// TIA Portal project "Arenas_Pantoja_Ospina_PF" (V15)
// Vorlageprojekt für das Buch mit Zielsystem S7-1200

(* hardware
DEVICE "S7-1200-Station_1"  S7-1200 Station
   slot 0: "Baugruppenträger_0"  Rack  V1.0
   slot 1: "PLC_1"  CPU 1214C AC/DC/Rly  6ES7 214-1BG40-0XB0  V4.1
*)

// ===== PLC "PLC_1"  CPU 1214C AC/DC/Rly =====

VAR_GLOBAL   // PLC tag table "Standard-Variablentabelle"
   "START" AT %E0.0 : Bool;
   "M200" AT %M200.0 : Bool;
   "P0" AT %M0.0 : Bool;
   "AUTOMATICO" AT %I6.0 : Bool;
   "MANUAL" AT %I6.1 : Bool;
   "P1" AT %M0.1 : Bool;
   "AAAAAAAAAAAAAAAAAAAAAAAAAAAAAAAAAAA" AT %M40.0 : Bool;
   "P2" AT %M0.2 : Bool;
   "I1_EntradaObjetos" AT %I0.1 : Bool;
   "P3" AT %M0.3 : Bool;
   "I2_SensorPasoInicial" AT %I0.2 : Bool;
   "FP_I2_SensorPasoInicial" AT %M50.0 : Bool;
   "P4" AT %M0.4 : Bool;
   "FN_I2_SensorPasoInicial" AT %M50.1 : Bool;
   "P5" AT %M0.5 : Bool;
   "I3_SensorVisionBR" AT %I0.3 : Bool;
   "I4_SensorVisionGR" AT %I0.4 : Bool;
   "I5_SensorVisionBG" AT %I0.5 : Bool;
   "P6" AT %M0.6 : Bool;
   "I6_BandaBascula" AT %I0.6 : Bool;
   "FP_I6_BandaBascula(1)" AT %M50.2 : Bool;
   "P7" AT %M0.7 : Bool;
   "P8" AT %M1.0 : Bool;
   "FP_I8_SensorLeft" AT %M50.3 : Bool;
   "I8_SensorLeft" AT %I1.0 : Bool;
   "FN_I8_SensorLeft" AT %M50.4 : Bool;
   "P9" AT %M1.1 : Bool;
   "P10" AT %M1.2 : Bool;
   "FP_I6_BandaBascula_2" AT %M50.5 : Bool;
   "P11" AT %M1.3 : Bool;
   "I7_SensorForward" AT %I0.7 : Bool;
   "FP_I7_SensorForward" AT %M50.6 : Bool;
   "P12" AT %M1.4 : Bool;
   "FN_I7_SensorForward_3" AT %M50.7 : Bool;
   "P13" AT %M1.5 : Bool;
   "P14" AT %M1.6 : Bool;
   "FP_I6_BandaBascula_3" AT %M51.0 : Bool;
   "P15" AT %M1.7 : Bool;
   "I9_SensorRigth" AT %I1.1 : Bool;
   "P16" AT %M2.0 : Bool;
   "FP_I9_SensorRigth" AT %M51.1 : Bool;
   "FN_I9_SensorRigth_2" AT %M51.2 : Bool;
   "P17" AT %M2.1 : Bool;
   "Q0_EntradaObjetos" AT %Q0.0 : Bool;
   "Q1_BandaInicial" AT %Q0.1 : Bool;
   "Q2_BandaInicial2" AT %Q0.2 : Bool;
   "Q3_Forward" AT %Q0.3 : Bool;
   "Q4_Left" AT %Q0.4 : Bool;
   "Q5_Right" AT %Q0.5 : Bool;
   "Q6_BandaLeft1" AT %Q0.6 : Bool;
   "Q7_BandaForward1" AT %Q0.7 : Bool;
   "Q8_BandaRigth1" AT %Q1.0 : Bool;
   "Tag_2" AT %MD0 : DWord;
   "I10_SensorLeft2" AT %I1.2 : Bool;
   "FP_I10_SensorLeft2" AT %M51.3 : Bool;
   "P18" AT %M2.2 : Bool;
   "P19" AT %M2.3 : Bool;
   "FN_I10_SensorLeft2" AT %M51.4 : Bool;
   "P20" AT %M2.4 : Bool;
   "I13_SensorLeft3" AT %I1.5 : Bool;
   "FP_I13_SensorLeft3" AT %M51.5 : Bool;
   "FN_I13_SensorLeft3" AT %M51.6 : Bool;
   "P21" AT %M2.5 : Bool;
   "P22" AT %M2.6 : Bool;
   "I11_SensorForward2" AT %I1.3 : Bool;
   "FP_I11_SensorForward2" AT %M51.7 : Bool;
   "P23" AT %M2.7 : Bool;
   "FN_I11_SensorForward2" AT %M52.0 : Bool;
   "P24" AT %M3.0 : Bool;
   "I14_SensorForward3" AT %I1.6 : Bool;
   "FP_I14_SensorForward3" AT %M52.1 : Bool;
   "P25" AT %M3.1 : Bool;
   "I12_SensorRigth2" AT %I1.4 : Bool;
   "FP_I12_SensorRigth2" AT %M52.2 : Bool;
   "P26" AT %M3.2 : Bool;
   "FN_I12_SensorRigth2" AT %M52.3 : Bool;
   "P27" AT %M3.3 : Bool;
   "P28" AT %M3.4 : Bool;
   "I15_SensorRigth3" AT %I1.7 : Bool;
   "FP_I15_SensorRigth3" AT %M52.4 : Bool;
   "P29" AT %M3.5 : Bool;
   "FN_I15_SensorRigth3" AT %M52.5 : Bool;
   "Q9_BandaLeft2" AT %Q1.1 : Bool;
   "Q10_BandaForward2" AT %Q1.2 : Bool;
   "Q11_BandaRigtht2" AT %Q1.3 : Bool;
   "Q12_BandaLeft3" AT %Q1.4 : Bool;
   "Q13_BandaForward3" AT %Q1.5 : Bool;
   "Q14_BandaRigth3" AT %Q1.6 : Bool;
   "Q17_PickZ1" AT %Q2.1 : Bool;
   "Q20_PickZ2" AT %Q2.4 : Bool;
   "Q23_PickZ3" AT %Q2.7 : Bool;
   "FN_I14_SensorForward3" AT %M52.6 : Bool;
   "P30" AT %M3.6 : Bool;
   "I16_SensorGrab1" AT %I2.0 : Bool;
   "FP_I16_SensorGrab1" AT %M52.7 : Bool;
   "P31" AT %M3.7 : Bool;
   "P32" AT %M4.0 : Bool;
   "P33" AT %M4.1 : Bool;
   "P34" AT %M4.2 : Bool;
   "P35" AT %M4.3 : Bool;
   "Q15_PickX1" AT %Q1.7 : Bool;
   "Q16_PickGrab1" AT %Q2.0 : Bool;
   "I17_SensorGrab2" AT %I2.1 : Bool;
   "FP_I17_SensorGrab1" AT %M53.0 : Bool;
   "P36" AT %M4.4 : Bool;
   "P37" AT %M4.5 : Bool;
   "P38" AT %M4.6 : Bool;
   "P39" AT %M4.7 : Bool;
   "P40" AT %M5.0 : Bool;
   "P41" AT %M5.1 : Bool;
   "Q18_PickX2" AT %Q2.2 : Bool;
   "Q19_PickGrab2" AT %Q2.3 : Bool;
   "I18_SensorGrab3" AT %I2.2 : Bool;
   "FP_I18_SensorGrab3" AT %M53.1 : Bool;
   "P42" AT %M5.2 : Bool;
   "P43" AT %M5.3 : Bool;
   "P44" AT %M5.4 : Bool;
   "P45" AT %M5.5 : Bool;
   "P46" AT %M5.6 : Bool;
   "P47" AT %M5.7 : Bool;
   "Q21_PickX3" AT %Q2.5 : Bool;
   "Q22_PickGrab3" AT %Q2.6 : Bool;
   "I19_SensorBandaA1" AT %I2.3 : Bool;
   "FP_I19_SensorBandaA1" AT %M53.2 : Bool;
   "P48" AT %M6.0 : Bool;
   "I20_SensorBandaA2" AT %I2.4 : Bool;
   "FP_I20_SensorBandaA2" AT %M53.3 : Bool;
   "P49" AT %M6.1 : Bool;
   "I21_SensorBandaA3" AT %I2.5 : Bool;
   "FP_21_SensorBandaA3" AT %M53.4 : Bool;
   "P50" AT %M6.2 : Bool;
   "Q24_BandaLeftA1" AT %Q3.0 : Bool;
   "Q25_BandaLeftA2" AT %Q3.1 : Bool;
   "Q26_BandaForwardA1" AT %Q3.2 : Bool;
   "Q27_BandaForwardA2" AT %Q3.3 : Bool;
   "Q28_BandaRightA1" AT %Q3.4 : Bool;
   "Q29_BandaRightA2" AT %Q3.5 : Bool;
   "Q30_EmisorA1" AT %Q3.6 : Bool;
   "Q31_EmisorA2" AT %Q3.7 : Bool;
   "Q32_EmisorA3" AT %Q4.0 : Bool;
   "P51" AT %M6.3 : Bool;
   "I22_LimAdelaA1" AT %I2.6 : Bool;
   "FP_I22_LimAdelaA1" AT %M53.5 : Bool;
   "P52" AT %M6.4 : Bool;
   "I23_LimSubA1" AT %I2.7 : Bool;
   "FP_I23_LimSubA1" AT %M53.6 : Bool;
   "Q33_AdelanteA1" AT %Q4.1 : Bool;
   "Q34_SubirA1" AT %Q4.2 : Bool;
   "P53" AT %M6.5 : Bool;
   "I24_LimAdelaA2" AT %I3.0 : Bool;
   "FP_I24_LimAdelaA2" AT %M53.7 : Bool;
   "P54" AT %M6.6 : Bool;
   "I25_LimSubA2" AT %I3.1 : Bool;
   "FN_I25_LimSubA2" AT %M54.0 : Bool;
   "Q36_AdelanteA2" AT %Q4.4 : Bool;
   "Q37_SubirA2" AT %Q4.5 : Bool;
   "P55" AT %M6.7 : Bool;
   "P56" AT %M7.0 : Bool;
   "Q39_AdelanteA3" AT %Q4.7 : Bool;
   "Q40_SubirA3" AT %Q5.0 : Bool;
   "P57" AT %M7.1 : Bool;
   "P58" AT %M7.2 : Bool;
   "P59" AT %M7.3 : Bool;
   "Right count" AT %QW40 : Int;
   "Tag_4" AT %QW50 : Int;
   "Q41_PosicionA1" AT %QW30 : Int;
   "Tag_6" AT %QW60 : Int;
   "Tag_7" AT %QW90 : Int;
   "Q42_PosicionA2" AT %QW32 : Int;
   "Tag_9" AT %QW33 : Int;
   "Q43_PosicionA3" AT %QW34 : Int;
   "P60" AT %M7.4 : Bool;
   "P61" AT %M7.5 : Bool;
   "P62" AT %M7.6 : Bool;
   "Q35_AtrasA1" AT %Q4.3 : Bool;
   "P63" AT %M7.7 : Bool;
   "P64" AT %M8.0 : Bool;
   "P65" AT %M8.1 : Bool;
   "P66" AT %M8.2 : Bool;
   "P67" AT %M8.3 : Bool;
   "Q38_AtrasA2" AT %Q4.6 : Bool;
   "P68" AT %M8.4 : Bool;
   "P69" AT %M8.5 : Bool;
   "P70" AT %M8.6 : Bool;
   "P71" AT %M8.7 : Bool;
   "Q41_AtrasA3" AT %Q5.1 : Bool;
   "I_4.0_PosicionA1" AT %I4.0 : Bool;
   "FN_I_4.0_PosicionA1" AT %M540.1 : Bool;
   "I_4.1_PosicionA2" AT %I4.1 : Bool;
   "FN_I_4.0_PosicionA1(1)" AT %M54.1 : Bool;
   "FN_I_4.1_PosicionA2" AT %M54.2 : Bool;
   "I_4.2_PosicionA3" AT %I4.2 : Bool;
   "FN_I_4.2_PosicionA3" AT %M54.3 : Bool;
   "P80" AT %M9.0 : Bool;
   "Left count" AT %QW36 : Word;
   "Forward count" AT %QW38 : Int;
   "M.Emitter" AT %I3.2 : Bool;
   "M.BI_B2" AT %I3.3 : Bool;
   "M.Q3_ON" AT %I3.4 : Bool;
   "M.Q3_OFF" AT %I3.5 : Bool;
   "M.LEFT_DECISION" AT %I3.6 : Bool;
   "M.RIGHT_DECISION" AT %I3.7 : Bool;
   "M.Left bands" AT %I4.3 : Bool;
   "M.Forward bands" AT %I4.4 : Bool;
   "M.Right bands" AT %I4.5 : Bool;
   "STOP" AT %I5.7 : Bool;
   "I4.6_M.GrabOn" AT %I4.6 : Bool;
   "I4.7_M.GrabOff" AT %I4.7 : Bool;
   "I5.0_M.EjeXOn" AT %I5.0 : Bool;
   "I5.2_M.EjezOn" AT %I5.2 : Bool;
   "I5.4_M.EmitterM" AT %I5.4 : Bool;
   "I5.1_M.EjeXOff" AT %I5.1 : Bool;
   "I5.3_M.EjezOff" AT %I5.3 : Bool;
   "Q44_LightAutomatico" AT %Q5.2 : Bool;
   "Q45_LightManual" AT %Q5.3 : Bool;
   "I5.5_M.BandasA" AT %I5.5 : Bool;
   "Q46.RemoverM" AT %Q5.4 : Bool;
   "Pin_BL" AT %M10.0 : Bool;
   "ENABLE_BL" AT %M15.0 : Bool;
   "M_Q2_B_LEFT" AT %M20.1 : Bool;
   "M_Q3_B_LEFT" AT %M20.2 : Bool;
   "M_Q4_B_LEFT" AT %M20.3 : Bool;
   "M_Q6_B_LEFT" AT %M20.5 : Bool;
   "M_Q9_B_LEFT" AT %M21.0 : Bool;
   "M_Q12_B_LEFT" AT %M21.3 : Bool;
   "Pout_BL" AT %M10.1 : Bool;
   "Pin_PL" AT %M10.2 : Bool;
   "ENABLE_PL" AT %M15.1 : Bool;
   "M_Q5_B_RIGHT" AT %M20.4 : Bool;
   "M_Q7" AT %M20.6 : Bool;
   "M_Q8_B_RIGHT" AT %M20.7 : Bool;
   "M_Q10" AT %M21.1 : Bool;
   "M_Q11_B_RIGHT" AT %M21.2 : Bool;
   "M_Q13" AT %M21.4 : Bool;
   "M_Q14_B_RIGHT" AT %M21.5 : Bool;
   "M_Q15_P_LEFT" AT %M21.6 : Bool;
   "M_Q16_P_LEFT" AT %M21.7 : Bool;
   "M_Q17_P_LEFT" AT %M22.0 : Bool;
   "M_Q18_B_PF" AT %M22.1 : Bool;
   "M_Q19_B_PF" AT %M22.2 : Bool;
   "M_Q20_B_PF" AT %M22.3 : Bool;
   "M_Q21_P_RIGHT" AT %M22.4 : Bool;
   "M_Q22_P_RIGHT" AT %M22.5 : Bool;
   "M_Q23_P_RIGHT" AT %M22.6 : Bool;
   "M_Q24_G_LEFT" AT %M22.7 : Bool;
   "M_Q25_G_LEFT" AT %M23.0 : Bool;
   "M_Q26_GF" AT %M23.1 : Bool;
   "M_Q27_GF" AT %M23.2 : Bool;
   "M_Q28" AT %M23.3 : Bool;
   "M_Q29" AT %M23.4 : Bool;
   "M_Q30_P_LEFT" AT %M23.5 : Bool;
   "Pout_PL" AT %M10.3 : Bool;
   "P52_Out" AT %M25.0 : Bool;
   "Pin_GL" AT %M10.4 : Bool;
   "ENABLE_GL" AT %M15.2 : Bool;
   "Pout_GL" AT %M10.5 : Bool;
   "M_Q31_B_PF" AT %M23.6 : Bool;
   "M_Q32_P_RIGHT" AT %M23.7 : Bool;
   "M_Q33_G_LEFT" AT %M24.0 : Bool;
   "M_Q34_G_LEFT" AT %M24.1 : Bool;
   "M_Q35_G_LEFT" AT %M24.2 : Bool;
   "M_Q36_GF" AT %M24.3 : Bool;
   "M_Q37_GF" AT %M24.4 : Bool;
   "M_Q38_GF" AT %M24.5 : Bool;
   "M_Q39" AT %M24.6 : Bool;
   "M_Q40" AT %M24.7 : Bool;
   "M_Q41_G_LEFT" AT %M26.0 : Bool;
   "M_Q42_G_FRONT" AT %M26.1 : Bool;
   "P57_Out" AT %M25.1 : Bool;
   "Pin_BF" AT %M10.6 : Bool;
   "ENABLE_BF" AT %M15.3 : Bool;
   "Pout_BF" AT %M10.7 : Bool;
   "M_Q2_B_FRONT" AT %M27.0 : Bool;
   "M_Q3_B_FRONT" AT %M27.1 : Bool;
   "NOHACENADA:D" AT %M27.2 : Bool;
   "M_Q7_B_FRONT" AT %M27.3 : Bool;
   "M_Q10_B_FRONT" AT %M27.4 : Bool;
   "M_Q13_B_FRONT" AT %M27.5 : Bool;
   "Pin_PF" AT %M11.0 : Bool;
   "ENABLE_PF" AT %M15.4 : Bool;
   "Pout_PF" AT %M11.1 : Bool;
   "Pin_GF" AT %M11.2 : Bool;
   "ENABLE_GF" AT %M15.5 : Bool;
   "Pout_GF" AT %M11.3 : Bool;
   "P54_Out" AT %M25.2 : Bool;
   "P58_Out" AT %M25.3 : Bool;
   "ENABLE_BR" AT %M15.6 : Bool;
   "Pin_BR" AT %M11.4 : Bool;
   "Pout_BR" AT %M11.5 : Bool;
   "M_Q2_B_RIGHT" AT %M27.6 : Bool;
   "M_Q3_B_RIGHT" AT %M27.7 : Bool;
   "Pin_PR" AT %M11.6 : Bool;
   "ENABLE_PR" AT %M15.7 : Bool;
   "Pout_PR" AT %M11.7 : Bool;
   "Pin_GR" AT %M12.0 : Bool;
   "ENABLE_GR" AT %M16.0 : Bool;
   "Pout_GR" AT %M12.1 : Bool;
   "P56_Out" AT %M25.4 : Bool;
   "P59_Out" AT %M25.5 : Bool;
   "M_Q41_GR" AT %M26.2 : Bool;
   "Tag_3" AT %M26.3 : Bool;
   "M_Q43_G_RIGHT" AT %M26.4 : Bool;
   "QR_LEFT" AT %M28.0 : Bool;
   "QR_FRONT" AT %M28.1 : Bool;
   "QR_RIGHT" AT %M28.2 : Bool;
   "Tag_5" AT %MD4 : DWord;
   "Tag_8" AT %MD8 : DWord;
   "Tag_10" AT %MD12 : DWord;
   "Tag_11" AT %MD16 : DWord;
   "Tag_12" AT %MD20 : DWord;
   "Tag_13" AT %MD24 : DWord;
   "Tag_14" AT %M40.1 : Bool;
   "fin_ciclo" AT %I6.2 : Bool;
   "fin_de_cilco" AT %M40.2 : Bool;
   "SensorVision_FLeft_1" AT %I6.3 : Bool;
   "SensorVision_FLeft_2" AT %I6.4 : Bool;
   "SensorVision_FForward_1" AT %I6.5 : Bool;
   "SensorVision_FForward_2" AT %I6.6 : Bool;
   "SensorVision_FRight_1" AT %I6.7 : Bool;
   "SensorVision_FRight_2" AT %I7.0 : Bool;
   "tiempoRecorrido" AT %M60.0 : Bool;
END_VAR

DATA_BLOCK "G_LEFT"   // DB1
{ S7_Optimized_Access := 'TRUE' }
VERSION : 0.1
// stored: InstanceOfName Grua
"Grua"
BEGIN
END_DATA_BLOCK

DATA_BLOCK "B_FRONT"   // DB3
{ S7_Optimized_Access := 'TRUE' }
VERSION : 0.1
// stored: InstanceOfName Bandas
"Bandas"
BEGIN
END_DATA_BLOCK

DATA_BLOCK "P_FRONT"   // DB4
{ S7_Optimized_Access := 'TRUE' }
VERSION : 0.1
// stored: InstanceOfName PickAndPlace
"PickAndPlace"
BEGIN
END_DATA_BLOCK

DATA_BLOCK "G_FRONT"   // DB5
{ S7_Optimized_Access := 'TRUE' }
VERSION : 0.1
// stored: InstanceOfName Grua
"Grua"
BEGIN
END_DATA_BLOCK

DATA_BLOCK "P_RIGHT"   // DB6
{ S7_Optimized_Access := 'TRUE' }
VERSION : 0.1
// stored: InstanceOfName PickAndPlace
"PickAndPlace"
BEGIN
END_DATA_BLOCK

DATA_BLOCK "G_RIGHT"   // DB7
{ S7_Optimized_Access := 'TRUE' }
VERSION : 0.1
// stored: InstanceOfName Grua
"Grua"
BEGIN
END_DATA_BLOCK

DATA_BLOCK "Datos_Ignition"   // DB9
{ S7_Optimized_Access := 'FALSE' }
VERSION : 0.1
   VAR
      START : Bool;
      MANUAL : Bool;
      STOP : Bool;
      AUTO : Bool;
      IGNI_FAC : Bool;
      F_1 : Bool;
      SF : Bool;   // Tag para la solución de la falla
      F_2_Left : Bool;
      F_2_Forward : Bool;
      F_2_Right : Bool;
      F_3_Left : Bool;
      F_3_Forward : Bool;
      F_3_Right : Bool;
      nPiezasAzules : Real;
      nPiezasAzules_I : Real;
      nPiezasVerdes : Real;
      nPiezasVerdes_I : Real;
      nPiezasVerdesTextura : Real;
      nPiezasVerdesTextura_I : Real;
      totalPiezas : Real;
      nPiezasDefectuosas_I : Real;
      nPiezasDefectuosas : Real;
      OEE_calidad : Real;
      tiempoProgramado : Real;
      tiempoEfectivo : Real;
      cantidadPiezasMOM : Real;
      OEE_disponibilidad : Real;
      OEE_desempeño : Real;
      OEE_global : Real;
      Macro_BL : Bool;
      Macro_PL : Bool;
      Macro_GL : Bool;
      Macro_BF : Bool;
      Macro_PF : Bool;
      Macro_GF : Bool;
      Macro_BR : Bool;
      Macro_PR : Bool;
      Macro_GR : Bool;
      MM_Emisor : Bool;
      MM_bandaInicial : Bool;
      MM_izquierda : Bool;
      MM_selectorRueda : Bool;
      MM_derecha : Bool;
      MM_bandasIzquierda : Bool;
      MM_bandasFrente : Bool;
      MM_bandasDercha : Bool;
      MM_agarrar : Bool;
      MM_ejeX : Bool;
      MM_ejeZ : Bool;
      MM_emisorCaja : Bool;
      MM_bandasRodillo : Bool;
   END_VAR
BEGIN
END_DATA_BLOCK

DATA_BLOCK "B_LEFT"   // DB28
{ S7_Optimized_Access := 'TRUE' }
VERSION : 0.1
// stored: InstanceOfName Bandas
"Bandas"
BEGIN
END_DATA_BLOCK

DATA_BLOCK "P_LEFT"   // DB46
{ S7_Optimized_Access := 'TRUE' }
VERSION : 0.1
// stored: InstanceOfName PickAndPlace
"PickAndPlace"
BEGIN
END_DATA_BLOCK

DATA_BLOCK "B_RIGHT"   // DB48
{ S7_Optimized_Access := 'TRUE' }
VERSION : 0.1
// stored: InstanceOfName Bandas
"Bandas"
BEGIN
END_DATA_BLOCK

// folder: System blocks/Program resources

DATA_BLOCK "T29"   // DB2
{ S7_Optimized_Access := 'TRUE' }
AUTHOR : Simatic
FAMILY : IEC
NAME : IEC_TMR
VERSION : 1.0
// stored: InstanceOfName IEC_TIMER
"IEC_TIMER"
BEGIN
END_DATA_BLOCK

DATA_BLOCK "C3_1"   // DB8
{ S7_Optimized_Access := 'TRUE' }
AUTHOR : Simatic
FAMILY : IEC
NAME : CNTR
VERSION : 1.0
// stored: InstanceOfName IEC_COUNTER
"IEC_COUNTER"
BEGIN
END_DATA_BLOCK

DATA_BLOCK "IEC_Timer_0_DB"   // DB10
{ S7_Optimized_Access := 'TRUE' }
AUTHOR : Simatic
FAMILY : IEC
NAME : IEC_TMR
VERSION : 1.0
// stored: InstanceOfName IEC_TIMER
"IEC_TIMER"
BEGIN
END_DATA_BLOCK

DATA_BLOCK "IEC_Timer_0_DB_1"   // DB11
{ S7_Optimized_Access := 'TRUE' }
AUTHOR : Simatic
FAMILY : IEC
NAME : IEC_TMR
VERSION : 1.0
// stored: InstanceOfName IEC_TIMER
"IEC_TIMER"
BEGIN
END_DATA_BLOCK

DATA_BLOCK "IEC_Timer_0_DB_2"   // DB12
{ S7_Optimized_Access := 'TRUE' }
AUTHOR : Simatic
FAMILY : IEC
NAME : IEC_TMR
VERSION : 1.0
// stored: InstanceOfName IEC_TIMER
"IEC_TIMER"
BEGIN
END_DATA_BLOCK

DATA_BLOCK "IEC_Timer_0_DB_3"   // DB13
{ S7_Optimized_Access := 'TRUE' }
AUTHOR : Simatic
FAMILY : IEC
NAME : IEC_TMR
VERSION : 1.0
// stored: InstanceOfName IEC_TIMER
"IEC_TIMER"
BEGIN
END_DATA_BLOCK

DATA_BLOCK "Counter_PDefectuosas"   // DB14
{ S7_Optimized_Access := 'TRUE' }
AUTHOR : Simatic
FAMILY : IEC
NAME : CNTR
VERSION : 1.0
// stored: InstanceOfName IEC_COUNTER
"IEC_COUNTER"
BEGIN
END_DATA_BLOCK

DATA_BLOCK "tiempoContado"   // DB15
{ S7_Optimized_Access := 'TRUE' }
AUTHOR : Simatic
FAMILY : IEC
NAME : IEC_TMR
VERSION : 1.0
// stored: InstanceOfName IEC_TIMER
"IEC_TIMER"
BEGIN
END_DATA_BLOCK

DATA_BLOCK "T16"   // DB16
{ S7_Optimized_Access := 'TRUE' }
AUTHOR : Simatic
FAMILY : IEC
NAME : IEC_TMR
VERSION : 1.0
// stored: InstanceOfName IEC_TIMER
"IEC_TIMER"
BEGIN
END_DATA_BLOCK

DATA_BLOCK "T17"   // DB17
{ S7_Optimized_Access := 'TRUE' }
AUTHOR : Simatic
FAMILY : IEC
NAME : IEC_TMR
VERSION : 1.0
// stored: InstanceOfName IEC_TIMER
"IEC_TIMER"
BEGIN
END_DATA_BLOCK

DATA_BLOCK "C"   // DB22
{ S7_Optimized_Access := 'TRUE' }
AUTHOR : Simatic
FAMILY : IEC
NAME : CNTR
VERSION : 1.0
// stored: InstanceOfName IEC_COUNTER
"IEC_COUNTER"
BEGIN
END_DATA_BLOCK

DATA_BLOCK "T22"   // DB25
{ S7_Optimized_Access := 'TRUE' }
AUTHOR : Simatic
FAMILY : IEC
NAME : IEC_TMR
VERSION : 1.0
// stored: InstanceOfName IEC_TIMER
"IEC_TIMER"
BEGIN
END_DATA_BLOCK

DATA_BLOCK "T26"   // DB29
{ S7_Optimized_Access := 'TRUE' }
AUTHOR : Simatic
FAMILY : IEC
NAME : IEC_TMR
VERSION : 1.0
// stored: InstanceOfName IEC_TIMER
"IEC_TIMER"
BEGIN
END_DATA_BLOCK

DATA_BLOCK "T27"   // DB30
{ S7_Optimized_Access := 'TRUE' }
AUTHOR : Simatic
FAMILY : IEC
NAME : IEC_TMR
VERSION : 1.0
// stored: InstanceOfName IEC_TIMER
"IEC_TIMER"
BEGIN
END_DATA_BLOCK

DATA_BLOCK "T28"   // DB31
{ S7_Optimized_Access := 'TRUE' }
AUTHOR : Simatic
FAMILY : IEC
NAME : IEC_TMR
VERSION : 1.0
// stored: InstanceOfName IEC_TIMER
"IEC_TIMER"
BEGIN
END_DATA_BLOCK

DATA_BLOCK "TON1"   // DB32
{ S7_Optimized_Access := 'TRUE' }
AUTHOR : Simatic
FAMILY : IEC
NAME : IEC_TMR
VERSION : 1.0
// stored: InstanceOfName IEC_TIMER
"IEC_TIMER"
BEGIN
END_DATA_BLOCK

DATA_BLOCK "TON2"   // DB36
{ S7_Optimized_Access := 'TRUE' }
AUTHOR : Simatic
FAMILY : IEC
NAME : IEC_TMR
VERSION : 1.0
// stored: InstanceOfName IEC_TIMER
"IEC_TIMER"
BEGIN
END_DATA_BLOCK

DATA_BLOCK "TON3"   // DB43
{ S7_Optimized_Access := 'TRUE' }
AUTHOR : Simatic
FAMILY : IEC
NAME : IEC_TMR
VERSION : 1.0
// stored: InstanceOfName IEC_TIMER
"IEC_TIMER"
BEGIN
END_DATA_BLOCK

DATA_BLOCK "TON4"   // DB44
{ S7_Optimized_Access := 'TRUE' }
AUTHOR : Simatic
FAMILY : IEC
NAME : IEC_TMR
VERSION : 1.0
// stored: InstanceOfName IEC_TIMER
"IEC_TIMER"
BEGIN
END_DATA_BLOCK

DATA_BLOCK "TON6"   // DB45
{ S7_Optimized_Access := 'TRUE' }
AUTHOR : Simatic
FAMILY : IEC
NAME : IEC_TMR
VERSION : 1.0
// stored: InstanceOfName IEC_TIMER
"IEC_TIMER"
BEGIN
END_DATA_BLOCK

DATA_BLOCK "C2_1"   // DB47
{ S7_Optimized_Access := 'TRUE' }
AUTHOR : Simatic
FAMILY : IEC
NAME : CNTR
VERSION : 1.0
// stored: InstanceOfName IEC_COUNTER
"IEC_COUNTER"
BEGIN
END_DATA_BLOCK

// folder: (top level)

FUNCTION_BLOCK "Bandas"   // FB1, LAD
{ S7_Optimized_Access := 'TRUE' }
VERSION : 0.1
   VAR_INPUT
      I8_SensorLeft : Bool;
      I10_SensorLeft2 : Bool;
      I13_SensorLeft3 : Bool;
   END_VAR
   VAR_OUTPUT
      Q2 : Bool;
      Q3 : Bool;
      Q4 : Bool;
      Q6 : Bool;
      Q9 : Bool;
      Q12 : Bool;
   END_VAR
   VAR_IN_OUT
      Pin : Bool;
      Pout : Bool;
   END_VAR
   VAR
      P7 : Bool;
      P8 : Bool;
      P9 : Bool;
      P18 : Bool;
      P19 : Bool;
      P20 : Bool;
      FP_I8_SensorLeft : Bool;
      FN_I8_SensorLeft : Bool;
      FP_I10_SensorLeft2 : Bool;
      FN_I10_SensorLeft2 : Bool;
      FP_I13_SensorLeft3 : Bool;
      FN_I13_SensorLeft3 : Bool;
   END_VAR
   VAR_TEMP   // added for the SCL form of the ladder/FBD networks
      _w1 : Bool;
   END_VAR
BEGIN

REGION Network 1
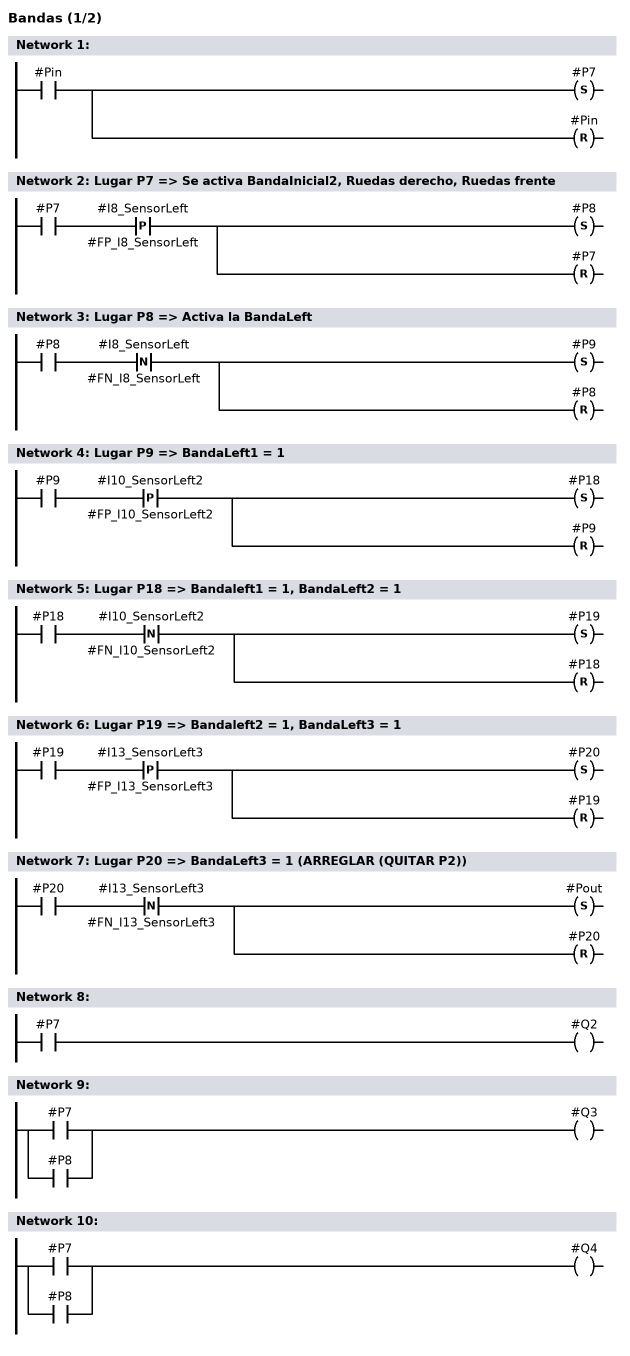
   RUNG wire#powerrail
      Contact( #Pin )
      wire#w1
      S_Coil( #P7 )
   END_RUNG
   RUNG wire#w1
      R_Coil( #Pin )
   END_RUNG
   // the same network as SCL:
   IF #Pin THEN
       #P7 := TRUE;
       #Pin := FALSE;
   END_IF;
END_REGION

REGION Network 2: Lugar P7 => Se activa BandaInicial2, Ruedas derecho, Ruedas frente
   RUNG wire#powerrail
      Contact( #P7 )
      P_Contact(operand := #I8_SensorLeft, bit := #FP_I8_SensorLeft)
      wire#w1
      S_Coil( #P8 )
   END_RUNG
   RUNG wire#w1
      R_Coil( #P7 )
   END_RUNG
   // the same network as SCL:
   #_w1 := #P7 AND #I8_SensorLeft AND NOT #FP_I8_SensorLeft;   // rising edge of #I8_SensorLeft
   #FP_I8_SensorLeft := #I8_SensorLeft;
   IF #_w1 THEN
       #P8 := TRUE;
       #P7 := FALSE;
   END_IF;
END_REGION

REGION Network 3: Lugar P8 => Activa la BandaLeft
   RUNG wire#powerrail
      Contact( #P8 )
      N_Contact(operand := #I8_SensorLeft, bit := #FN_I8_SensorLeft)
      wire#w1
      S_Coil( #P9 )
   END_RUNG
   RUNG wire#w1
      R_Coil( #P8 )
   END_RUNG
   // the same network as SCL:
   #_w1 := #P8 AND NOT #I8_SensorLeft AND #FN_I8_SensorLeft;   // falling edge of #I8_SensorLeft
   #FN_I8_SensorLeft := #I8_SensorLeft;
   IF #_w1 THEN
       #P9 := TRUE;
       #P8 := FALSE;
   END_IF;
END_REGION

REGION Network 4: Lugar P9 => BandaLeft1 = 1
   RUNG wire#powerrail
      Contact( #P9 )
      P_Contact(operand := #I10_SensorLeft2, bit := #FP_I10_SensorLeft2)
      wire#w1
      S_Coil( #P18 )
   END_RUNG
   RUNG wire#w1
      R_Coil( #P9 )
   END_RUNG
   // the same network as SCL:
   #_w1 := #P9 AND #I10_SensorLeft2 AND NOT #FP_I10_SensorLeft2;   // rising edge of #I10_SensorLeft2
   #FP_I10_SensorLeft2 := #I10_SensorLeft2;
   IF #_w1 THEN
       #P18 := TRUE;
       #P9 := FALSE;
   END_IF;
END_REGION

REGION Network 5: Lugar P18 => Bandaleft1 = 1, BandaLeft2 = 1
   RUNG wire#powerrail
      Contact( #P18 )
      N_Contact(operand := #I10_SensorLeft2, bit := #FN_I10_SensorLeft2)
      wire#w1
      S_Coil( #P19 )
   END_RUNG
   RUNG wire#w1
      R_Coil( #P18 )
   END_RUNG
   // the same network as SCL:
   #_w1 := #P18 AND NOT #I10_SensorLeft2 AND #FN_I10_SensorLeft2;   // falling edge of #I10_SensorLeft2
   #FN_I10_SensorLeft2 := #I10_SensorLeft2;
   IF #_w1 THEN
       #P19 := TRUE;
       #P18 := FALSE;
   END_IF;
END_REGION

REGION Network 6: Lugar P19 => Bandaleft2 = 1, BandaLeft3 = 1
   RUNG wire#powerrail
      Contact( #P19 )
      P_Contact(operand := #I13_SensorLeft3, bit := #FP_I13_SensorLeft3)
      wire#w1
      S_Coil( #P20 )
   END_RUNG
   RUNG wire#w1
      R_Coil( #P19 )
   END_RUNG
   // the same network as SCL:
   #_w1 := #P19 AND #I13_SensorLeft3 AND NOT #FP_I13_SensorLeft3;   // rising edge of #I13_SensorLeft3
   #FP_I13_SensorLeft3 := #I13_SensorLeft3;
   IF #_w1 THEN
       #P20 := TRUE;
       #P19 := FALSE;
   END_IF;
END_REGION

REGION Network 7: Lugar P20 => BandaLeft3 = 1 (ARREGLAR (QUITAR P2))
   RUNG wire#powerrail
      Contact( #P20 )
      N_Contact(operand := #I13_SensorLeft3, bit := #FN_I13_SensorLeft3)
      wire#w1
      S_Coil( #Pout )
   END_RUNG
   RUNG wire#w1
      R_Coil( #P20 )
   END_RUNG
   // the same network as SCL:
   #_w1 := #P20 AND NOT #I13_SensorLeft3 AND #FN_I13_SensorLeft3;   // falling edge of #I13_SensorLeft3
   #FN_I13_SensorLeft3 := #I13_SensorLeft3;
   IF #_w1 THEN
       #Pout := TRUE;
       #P20 := FALSE;
   END_IF;
END_REGION

REGION Network 8
   RUNG wire#powerrail
      Contact( #P7 )
      Coil( #Q2 )
   END_RUNG
   // the same network as SCL:
   #Q2 := #P7;
END_REGION

REGION Network 9
   RUNG wire#powerrail
      Contact( #P7 )
      wire#w1
      Coil( #Q3 )
   END_RUNG
   RUNG wire#powerrail
      Contact( #P8 )
   END_RUNG wire#w1
   // the same network as SCL:
   #Q3 := #P7 OR #P8;
END_REGION

REGION Network 10
   RUNG wire#powerrail
      Contact( #P7 )
      wire#w1
      Coil( #Q4 )
   END_RUNG
   RUNG wire#powerrail
      Contact( #P8 )
   END_RUNG wire#w1
   // the same network as SCL:
   #Q4 := #P7 OR #P8;
END_REGION

REGION Network 11
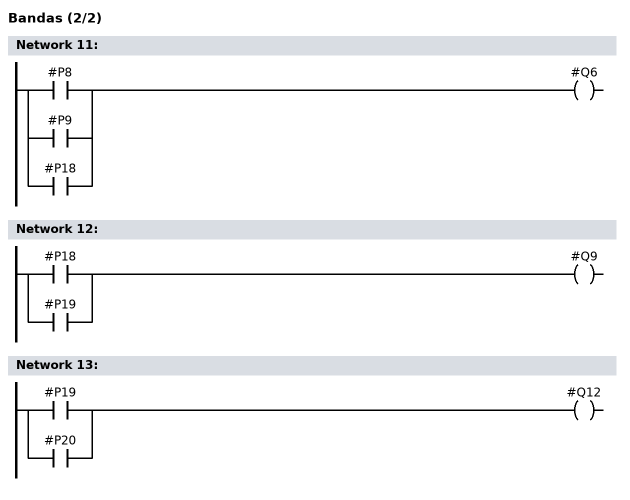
   RUNG wire#powerrail
      Contact( #P8 )
      wire#w1
      Coil( #Q6 )
   END_RUNG
   RUNG wire#powerrail
      Contact( #P9 )
   END_RUNG wire#w1
   RUNG wire#powerrail
      Contact( #P18 )
   END_RUNG wire#w1
   // the same network as SCL:
   #Q6 := #P8 OR #P9 OR #P18;
END_REGION

REGION Network 12
   RUNG wire#powerrail
      Contact( #P18 )
      wire#w1
      Coil( #Q9 )
   END_RUNG
   RUNG wire#powerrail
      Contact( #P19 )
   END_RUNG wire#w1
   // the same network as SCL:
   #Q9 := #P18 OR #P19;
END_REGION

REGION Network 13
   RUNG wire#powerrail
      Contact( #P19 )
      wire#w1
      Coil( #Q12 )
   END_RUNG
   RUNG wire#powerrail
      Contact( #P20 )
   END_RUNG wire#w1
   // the same network as SCL:
   #Q12 := #P19 OR #P20;
END_REGION
END_FUNCTION_BLOCK

FUNCTION_BLOCK "PickAndPlace"   // FB2, LAD
{ S7_Optimized_Access := 'TRUE' }
VERSION : 0.1
   VAR_INPUT
      I16_SensorGrab1 : Bool;
   END_VAR
   VAR_OUTPUT
      Q15 : Bool;
      Q16 : Bool;
      Q17 : Bool;
      Q30 : Bool;
   END_VAR
   VAR_IN_OUT
      Pin_PL : Bool;
      Pout_PL : Bool;
   END_VAR
   VAR
      P21 : Bool;
      P30 : Bool;
      P31 : Bool;
      P32 : Bool;
      P33 : Bool;
      P34 : Bool;
      P35 : Bool;
      FP_I16_SensorGrab1 : Bool;
   END_VAR
   VAR_TEMP   // added for the SCL form of the ladder/FBD networks
      _w1 : Bool;
   END_VAR
BEGIN

REGION Network 1
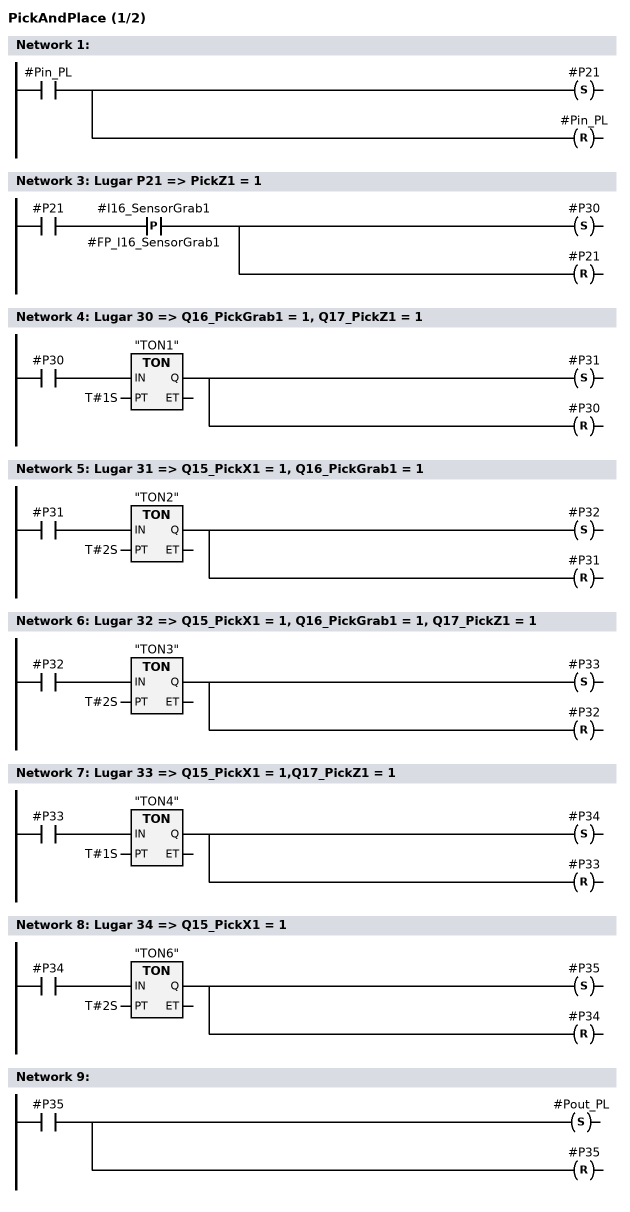
   RUNG wire#powerrail
      Contact( #Pin_PL )
      wire#w1
      S_Coil( #P21 )
   END_RUNG
   RUNG wire#w1
      R_Coil( #Pin_PL )
   END_RUNG
   // the same network as SCL:
   IF #Pin_PL THEN
       #P21 := TRUE;
       #Pin_PL := FALSE;
   END_IF;
END_REGION

REGION Network 3: Lugar P21 => PickZ1 = 1
   RUNG wire#powerrail
      Contact( #P21 )
      P_Contact(operand := #I16_SensorGrab1, bit := #FP_I16_SensorGrab1)
      wire#w1
      S_Coil( #P30 )
   END_RUNG
   RUNG wire#w1
      R_Coil( #P21 )
   END_RUNG
   // the same network as SCL:
   #_w1 := #P21 AND #I16_SensorGrab1 AND NOT #FP_I16_SensorGrab1;   // rising edge of #I16_SensorGrab1
   #FP_I16_SensorGrab1 := #I16_SensorGrab1;
   IF #_w1 THEN
       #P30 := TRUE;
       #P21 := FALSE;
   END_IF;
END_REGION

REGION Network 4: Lugar 30 => Q16_PickGrab1 = 1, Q17_PickZ1 = 1
   "TON1".TON(IN := #P30, PT := T#1S);
   IF "TON1".Q THEN
       #P31 := TRUE;
       #P30 := FALSE;
   END_IF;
END_REGION

REGION Network 5: Lugar 31 => Q15_PickX1 = 1, Q16_PickGrab1 = 1
   "TON2".TON(IN := #P31, PT := T#2S);
   IF "TON2".Q THEN
       #P32 := TRUE;
       #P31 := FALSE;
   END_IF;
END_REGION

REGION Network 6: Lugar 32 => Q15_PickX1 = 1, Q16_PickGrab1 = 1, Q17_PickZ1 = 1
   "TON3".TON(IN := #P32, PT := T#2S);
   IF "TON3".Q THEN
       #P33 := TRUE;
       #P32 := FALSE;
   END_IF;
END_REGION

REGION Network 7: Lugar 33 => Q15_PickX1 = 1,Q17_PickZ1 = 1
   "TON4".TON(IN := #P33, PT := T#1S);
   IF "TON4".Q THEN
       #P34 := TRUE;
       #P33 := FALSE;
   END_IF;
END_REGION

REGION Network 8: Lugar 34 => Q15_PickX1 = 1
   "TON6".TON(IN := #P34, PT := T#2S);
   IF "TON6".Q THEN
       #P35 := TRUE;
       #P34 := FALSE;
   END_IF;
END_REGION

REGION Network 9
   RUNG wire#powerrail
      Contact( #P35 )
      wire#w1
      S_Coil( #Pout_PL )
   END_RUNG
   RUNG wire#w1
      R_Coil( #P35 )
   END_RUNG
   // the same network as SCL:
   IF #P35 THEN
       #Pout_PL := TRUE;
       #P35 := FALSE;
   END_IF;
END_REGION

REGION Network 10
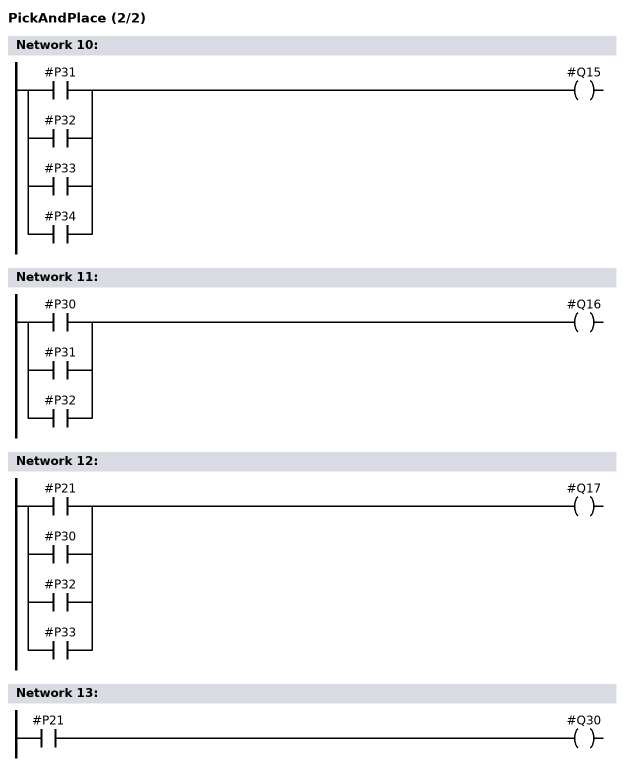
   RUNG wire#powerrail
      Contact( #P31 )
      wire#w1
      Coil( #Q15 )
   END_RUNG
   RUNG wire#powerrail
      Contact( #P32 )
   END_RUNG wire#w1
   RUNG wire#powerrail
      Contact( #P33 )
   END_RUNG wire#w1
   RUNG wire#powerrail
      Contact( #P34 )
   END_RUNG wire#w1
   // the same network as SCL:
   #Q15 := #P31 OR #P32 OR #P33 OR #P34;
END_REGION

REGION Network 11
   RUNG wire#powerrail
      Contact( #P30 )
      wire#w1
      Coil( #Q16 )
   END_RUNG
   RUNG wire#powerrail
      Contact( #P31 )
   END_RUNG wire#w1
   RUNG wire#powerrail
      Contact( #P32 )
   END_RUNG wire#w1
   // the same network as SCL:
   #Q16 := #P30 OR #P31 OR #P32;
END_REGION

REGION Network 12
   RUNG wire#powerrail
      Contact( #P21 )
      wire#w1
      Coil( #Q17 )
   END_RUNG
   RUNG wire#powerrail
      Contact( #P30 )
   END_RUNG wire#w1
   RUNG wire#powerrail
      Contact( #P32 )
   END_RUNG wire#w1
   RUNG wire#powerrail
      Contact( #P33 )
   END_RUNG wire#w1
   // the same network as SCL:
   #Q17 := #P21 OR #P30 OR #P32 OR #P33;
END_REGION

REGION Network 13
   RUNG wire#powerrail
      Contact( #P21 )
      Coil( #Q30 )
   END_RUNG
   // the same network as SCL:
   #Q30 := #P21;
END_REGION
END_FUNCTION_BLOCK

FUNCTION_BLOCK "Grua"   // FB3, LAD
{ S7_Optimized_Access := 'TRUE' }
VERSION : 0.1
   VAR_INPUT
      I19_SensorBandaA1 : Bool;
      "I_4.0_PosicionA1" : Bool;
   END_VAR
   VAR_OUTPUT
      P52_Out : Bool;
      Q24 : Bool;
      Q25 : Bool;
      Q33 : Bool;
      Q34 : Bool;
      Q35 : Bool;
      Q41 : Bool;
      P57_Out : Bool;
   END_VAR
   VAR_IN_OUT
      Pin_GL : Bool;
      Pout_GL : Bool;
   END_VAR
   VAR
      P35 : Bool;
      P48 : Bool;
      P51 : Bool;
      P52 : Bool;
      P57 : Bool;
      P60 : Bool;
      P61 : Bool;
      P62 : Bool;
      P63 : Bool;
      FP_I19_SensorBandaA1 : Bool;
      "FN_I_4.0_PosicionA1" : Bool;
   END_VAR
   VAR_TEMP   // added for the SCL form of the ladder/FBD networks
      _w1 : Bool;
   END_VAR
BEGIN

REGION Network 2
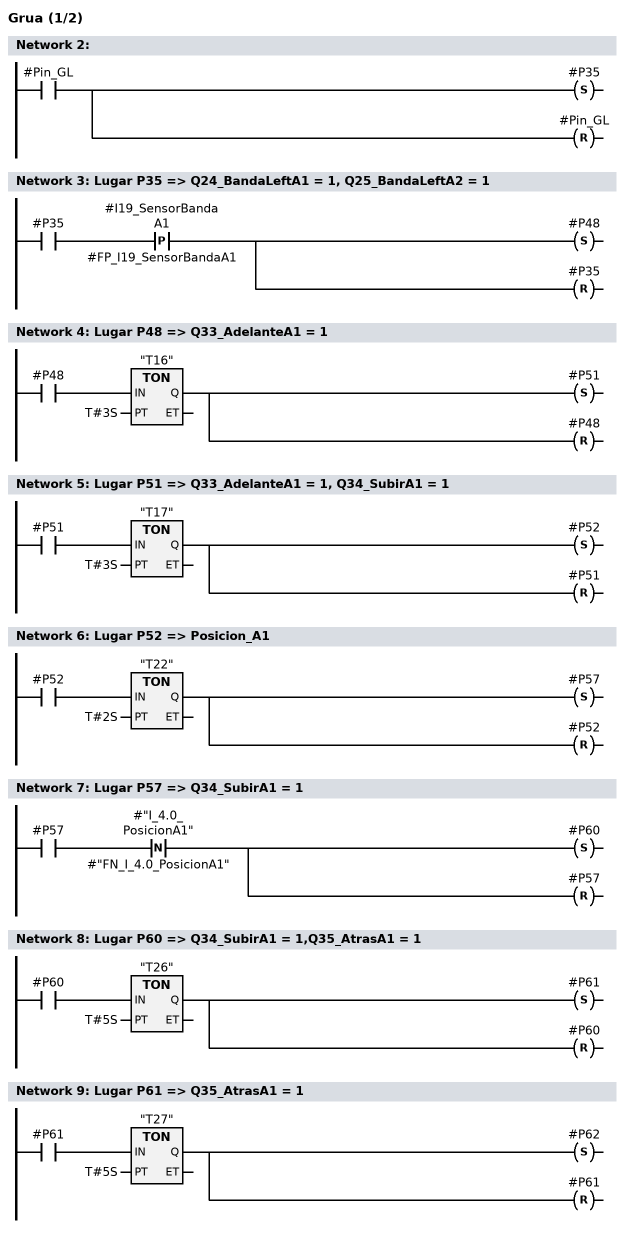
   RUNG wire#powerrail
      Contact( #Pin_GL )
      wire#w1
      S_Coil( #P35 )
   END_RUNG
   RUNG wire#w1
      R_Coil( #Pin_GL )
   END_RUNG
   // the same network as SCL:
   IF #Pin_GL THEN
       #P35 := TRUE;
       #Pin_GL := FALSE;
   END_IF;
END_REGION

REGION Network 3: Lugar P35 => Q24_BandaLeftA1 = 1, Q25_BandaLeftA2 = 1
   RUNG wire#powerrail
      Contact( #P35 )
      P_Contact(operand := #I19_SensorBandaA1, bit := #FP_I19_SensorBandaA1)
      wire#w1
      S_Coil( #P48 )
   END_RUNG
   RUNG wire#w1
      R_Coil( #P35 )
   END_RUNG
   // the same network as SCL:
   #_w1 := #P35 AND #I19_SensorBandaA1 AND NOT #FP_I19_SensorBandaA1;   // rising edge of #I19_SensorBandaA1
   #FP_I19_SensorBandaA1 := #I19_SensorBandaA1;
   IF #_w1 THEN
       #P48 := TRUE;
       #P35 := FALSE;
   END_IF;
END_REGION

REGION Network 4: Lugar P48 => Q33_AdelanteA1 = 1
   "T16".TON(IN := #P48, PT := T#3S);
   IF "T16".Q THEN
       #P51 := TRUE;
       #P48 := FALSE;
   END_IF;
END_REGION

REGION Network 5: Lugar P51 => Q33_AdelanteA1 = 1, Q34_SubirA1 = 1
   "T17".TON(IN := #P51, PT := T#3S);
   IF "T17".Q THEN
       #P52 := TRUE;
       #P51 := FALSE;
   END_IF;
END_REGION

REGION Network 6: Lugar P52 => Posicion_A1
   "T22".TON(IN := #P52, PT := T#2S);
   IF "T22".Q THEN
       #P57 := TRUE;
       #P52 := FALSE;
   END_IF;
END_REGION

REGION Network 7: Lugar P57 => Q34_SubirA1 = 1
   RUNG wire#powerrail
      Contact( #P57 )
      N_Contact(operand := #"I_4.0_PosicionA1", bit := #"FN_I_4.0_PosicionA1")
      wire#w1
      S_Coil( #P60 )
   END_RUNG
   RUNG wire#w1
      R_Coil( #P57 )
   END_RUNG
   // the same network as SCL:
   #_w1 := #P57 AND NOT #"I_4.0_PosicionA1" AND #"FN_I_4.0_PosicionA1";   // falling edge of #"I_4.0_PosicionA1"
   #"FN_I_4.0_PosicionA1" := #"I_4.0_PosicionA1";
   IF #_w1 THEN
       #P60 := TRUE;
       #P57 := FALSE;
   END_IF;
END_REGION

REGION Network 8: Lugar P60 => Q34_SubirA1 = 1,Q35_AtrasA1 = 1
   "T26".TON(IN := #P60, PT := T#5S);
   IF "T26".Q THEN
       #P61 := TRUE;
       #P60 := FALSE;
   END_IF;
END_REGION

REGION Network 9: Lugar P61 => Q35_AtrasA1 = 1
   "T27".TON(IN := #P61, PT := T#5S);
   IF "T27".Q THEN
       #P62 := TRUE;
       #P61 := FALSE;
   END_IF;
END_REGION

REGION Network 10: Lugar P62 => Memoria
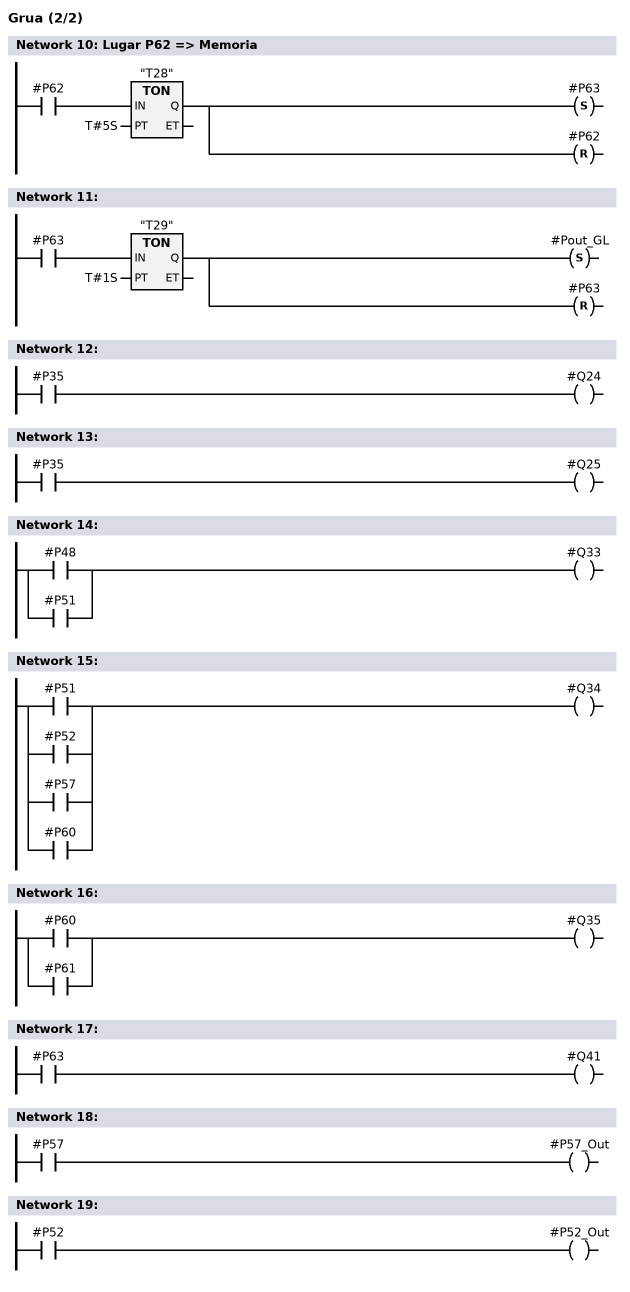
   "T28".TON(IN := #P62, PT := T#5S);
   IF "T28".Q THEN
       #P63 := TRUE;
       #P62 := FALSE;
   END_IF;
END_REGION

REGION Network 11
   "T29".TON(IN := #P63, PT := T#1S);
   IF "T29".Q THEN
       #Pout_GL := TRUE;
       #P63 := FALSE;
   END_IF;
END_REGION

REGION Network 12
   RUNG wire#powerrail
      Contact( #P35 )
      Coil( #Q24 )
   END_RUNG
   // the same network as SCL:
   #Q24 := #P35;
END_REGION

REGION Network 13
   RUNG wire#powerrail
      Contact( #P35 )
      Coil( #Q25 )
   END_RUNG
   // the same network as SCL:
   #Q25 := #P35;
END_REGION

REGION Network 14
   RUNG wire#powerrail
      Contact( #P48 )
      wire#w1
      Coil( #Q33 )
   END_RUNG
   RUNG wire#powerrail
      Contact( #P51 )
   END_RUNG wire#w1
   // the same network as SCL:
   #Q33 := #P48 OR #P51;
END_REGION

REGION Network 15
   RUNG wire#powerrail
      Contact( #P51 )
      wire#w1
      Coil( #Q34 )
   END_RUNG
   RUNG wire#powerrail
      Contact( #P52 )
   END_RUNG wire#w1
   RUNG wire#powerrail
      Contact( #P57 )
   END_RUNG wire#w1
   RUNG wire#powerrail
      Contact( #P60 )
   END_RUNG wire#w1
   // the same network as SCL:
   #Q34 := #P51 OR #P52 OR #P57 OR #P60;
END_REGION

REGION Network 16
   RUNG wire#powerrail
      Contact( #P60 )
      wire#w1
      Coil( #Q35 )
   END_RUNG
   RUNG wire#powerrail
      Contact( #P61 )
   END_RUNG wire#w1
   // the same network as SCL:
   #Q35 := #P60 OR #P61;
END_REGION

REGION Network 17
   RUNG wire#powerrail
      Contact( #P63 )
      Coil( #Q41 )
   END_RUNG
   // the same network as SCL:
   #Q41 := #P63;
END_REGION

REGION Network 18
   RUNG wire#powerrail
      Contact( #P57 )
      Coil( #P57_Out )
   END_RUNG
   // the same network as SCL:
   #P57_Out := #P57;
END_REGION

REGION Network 19
   RUNG wire#powerrail
      Contact( #P52 )
      Coil( #P52_Out )
   END_RUNG
   // the same network as SCL:
   #P52_Out := #P52;
END_REGION
END_FUNCTION_BLOCK

FUNCTION "MHJ-PLC-Lab-Function-S71200" : Void   // FC9000, SCL
{ S7_Optimized_Access := 'TRUE' }
VERSION : 0.1
   VAR_TEMP
      rdTimeReturn : Int;
      outputTime : DTL;
      SyncVal : Byte;
      forVal : Int;
      forVal_2 : Int;
      Value : Byte;
   END_VAR
   VAR CONSTANT
      CompVal : Byte := 16#34;
      Value_01 : Byte := 16#11;
      Value_01_DW : DWord := 16#A165_D992;
      Value_02_DW : DWord := 16#58BE_4401;
   END_VAR
BEGIN

   #Value:=PEEK(area := 16#82,
        dbNumber := 0,
        byteOffset := 511);
   #Value := #Value + 1;

   POKE(area := 16#82,
        dbNumber := 0,
        byteOffset := 511,
        value := #Value);

   POKE(area:=16#81,
        dbNumber:=0,
        byteOffset:=1016,
        value:=#Value_01_DW);
   POKE(area := 16#81,
        dbNumber := 0,
        byteOffset := 1020,
        value := #Value_02_DW);

   POKE(area := 16#81,
        dbNumber := 0,
        byteOffset := 511,
        value := B#16#00);

   FOR #forVal := 0 TO 120 DO
       FOR #forVal_2:=0 TO 10 DO
           #rdTimeReturn:=RD_SYS_T(#outputTime);
           #rdTimeReturn := WR_SYS_T(#outputTime);
           #rdTimeReturn := RD_SYS_T(#outputTime);
           #rdTimeReturn := WR_SYS_T(#outputTime);
       END_FOR;
       #SyncVal:= PEEK(area := 16#81,
                      dbNumber := 0,
                      byteOffset := 511);
       IF #SyncVal = #CompVal THEN
          GOTO M_1;
       END_IF;
   END_FOR;
   RETURN;

   M_1:
   POKE(area := 16#81,
        dbNumber := 0,
        byteOffset := 511,
        value := B#16#0);
END_FUNCTION

ORGANIZATION_BLOCK "Main"   // OB1, LAD, ProgramCycle
TITLE = "Main Program Sweep (Cycle)"
{ S7_Optimized_Access := 'TRUE' }
VERSION : 0.1
   VAR_INPUT
      Initial_Call : Bool;   // Initial call of this OB
      Remanence : Bool;   // =True, if remanent data are available
   END_VAR
   VAR_TEMP   // added for the SCL form of the ladder/FBD networks
      _w1 : Bool;
   END_VAR
BEGIN

REGION Network 1: Konnektierungsbaustein für PLC-Lab
   // Im Netzwerk 1 wird der Konnektierungsbaustein für PLC-Lab aufgerufen.
   // Dieser Aufruf darf nicht entfernt werden!
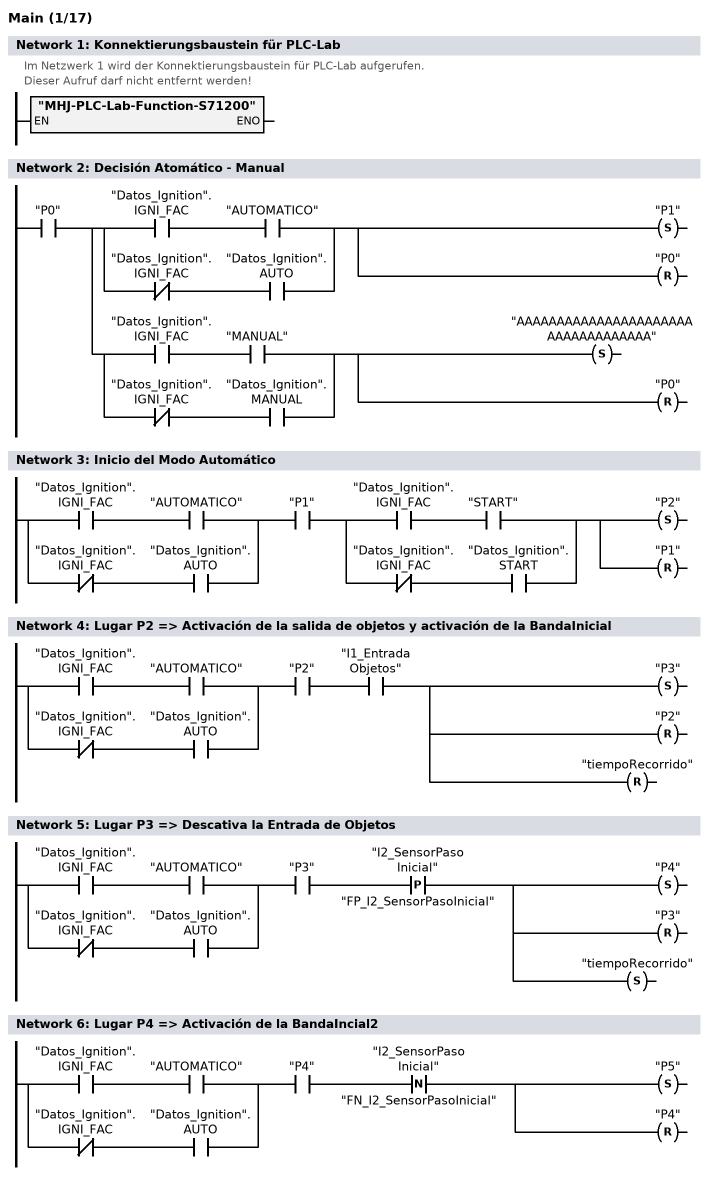
   RUNG wire#powerrail
      "MHJ-PLC-Lab-Function-S71200"()
   END_RUNG
   // the same network as SCL:
   "MHJ-PLC-Lab-Function-S71200"();
END_REGION

REGION Network 2: Decisión Atomático - Manual
   RUNG wire#powerrail
      Contact( "P0" )
      wire#w1
      Contact( "Datos_Ignition".IGNI_FAC )
      Contact( "AUTOMATICO" )
      wire#w2
      S_Coil( "P1" )
   END_RUNG
   RUNG wire#w1
      I_Contact( "Datos_Ignition".IGNI_FAC )
      Contact( "Datos_Ignition".AUTO )
   END_RUNG wire#w2
   RUNG wire#w2
      R_Coil( "P0" )
   END_RUNG
   RUNG wire#w1
      Contact( "Datos_Ignition".IGNI_FAC )
      Contact( "MANUAL" )
      wire#w3
      S_Coil( "AAAAAAAAAAAAAAAAAAAAAAAAAAAAAAAAAAA" )
   END_RUNG
   RUNG wire#w1
      I_Contact( "Datos_Ignition".IGNI_FAC )
      Contact( "Datos_Ignition".MANUAL )
   END_RUNG wire#w3
   RUNG wire#w3
      R_Coil( "P0" )
   END_RUNG
   // the same network as SCL:
   IF "P0" AND (("Datos_Ignition".IGNI_FAC AND "AUTOMATICO") OR (NOT "Datos_Ignition".IGNI_FAC AND "Datos_Ignition".AUTO)) THEN
       "P1" := TRUE;
   END_IF;
   #_w1 := "P0";
   IF "P0" AND (("Datos_Ignition".IGNI_FAC AND "AUTOMATICO") OR (NOT "Datos_Ignition".IGNI_FAC AND "Datos_Ignition".AUTO)) THEN
       "P0" := FALSE;
   END_IF;
   IF #_w1 AND (("Datos_Ignition".IGNI_FAC AND "MANUAL") OR (NOT "Datos_Ignition".IGNI_FAC AND "Datos_Ignition".MANUAL)) THEN
       "AAAAAAAAAAAAAAAAAAAAAAAAAAAAAAAAAAA" := TRUE;
       "P0" := FALSE;
   END_IF;
END_REGION

REGION Network 3: Inicio del Modo Automático
   RUNG wire#powerrail
      Contact( "Datos_Ignition".IGNI_FAC )
      Contact( "AUTOMATICO" )
      wire#w1
      Contact( "P1" )
      wire#w2
      Contact( "Datos_Ignition".IGNI_FAC )
      Contact( "START" )
      wire#w3
      S_Coil( "P2" )
   END_RUNG
   RUNG wire#powerrail
      I_Contact( "Datos_Ignition".IGNI_FAC )
      Contact( "Datos_Ignition".AUTO )
   END_RUNG wire#w1
   RUNG wire#w2
      I_Contact( "Datos_Ignition".IGNI_FAC )
      Contact( "Datos_Ignition".START )
   END_RUNG wire#w3
   RUNG wire#w3
      R_Coil( "P1" )
   END_RUNG
   // the same network as SCL:
   IF (("Datos_Ignition".IGNI_FAC AND "AUTOMATICO") OR (NOT "Datos_Ignition".IGNI_FAC AND "Datos_Ignition".AUTO)) AND "P1" AND (("Datos_Ignition".IGNI_FAC AND "START") OR (NOT "Datos_Ignition".IGNI_FAC AND "Datos_Ignition".START)) THEN
       "P2" := TRUE;
       "P1" := FALSE;
   END_IF;
END_REGION

REGION Network 4: Lugar P2 => Activación de la salida de objetos y activación de la BandaInicial
   RUNG wire#powerrail
      Contact( "Datos_Ignition".IGNI_FAC )
      Contact( "AUTOMATICO" )
      wire#w1
      Contact( "P2" )
      Contact( "I1_EntradaObjetos" )
      wire#w2
      S_Coil( "P3" )
   END_RUNG
   RUNG wire#powerrail
      I_Contact( "Datos_Ignition".IGNI_FAC )
      Contact( "Datos_Ignition".AUTO )
   END_RUNG wire#w1
   RUNG wire#w2
      R_Coil( "P2" )
   END_RUNG
   RUNG wire#w2
      R_Coil( "tiempoRecorrido" )
   END_RUNG
   // the same network as SCL:
   IF (("Datos_Ignition".IGNI_FAC AND "AUTOMATICO") OR (NOT "Datos_Ignition".IGNI_FAC AND "Datos_Ignition".AUTO)) AND "P2" AND "I1_EntradaObjetos" THEN
       "P3" := TRUE;
   END_IF;
   #_w1 := (("Datos_Ignition".IGNI_FAC AND "AUTOMATICO") OR (NOT "Datos_Ignition".IGNI_FAC AND "Datos_Ignition".AUTO)) AND "P2" AND "I1_EntradaObjetos";
   IF #_w1 THEN
       "P2" := FALSE;
       "tiempoRecorrido" := FALSE;
   END_IF;
END_REGION

REGION Network 5: Lugar P3 => Descativa la Entrada de Objetos
   RUNG wire#powerrail
      Contact( "Datos_Ignition".IGNI_FAC )
      Contact( "AUTOMATICO" )
      wire#w1
      Contact( "P3" )
      P_Contact(operand := "I2_SensorPasoInicial", bit := "FP_I2_SensorPasoInicial")
      wire#w2
      S_Coil( "P4" )
   END_RUNG
   RUNG wire#powerrail
      I_Contact( "Datos_Ignition".IGNI_FAC )
      Contact( "Datos_Ignition".AUTO )
   END_RUNG wire#w1
   RUNG wire#w2
      R_Coil( "P3" )
   END_RUNG
   RUNG wire#w2
      S_Coil( "tiempoRecorrido" )
   END_RUNG
   // the same network as SCL:
   #_w1 := (("Datos_Ignition".IGNI_FAC AND "AUTOMATICO") OR (NOT "Datos_Ignition".IGNI_FAC AND "Datos_Ignition".AUTO)) AND "P3" AND "I2_SensorPasoInicial" AND NOT "FP_I2_SensorPasoInicial";   // rising edge of "I2_SensorPasoInicial"
   "FP_I2_SensorPasoInicial" := "I2_SensorPasoInicial";
   IF #_w1 THEN
       "P4" := TRUE;
       "P3" := FALSE;
       "tiempoRecorrido" := TRUE;
   END_IF;
END_REGION

REGION Network 6: Lugar P4 => Activación de la BandaIncial2
   RUNG wire#powerrail
      Contact( "Datos_Ignition".IGNI_FAC )
      Contact( "AUTOMATICO" )
      wire#w1
      Contact( "P4" )
      N_Contact(operand := "I2_SensorPasoInicial", bit := "FN_I2_SensorPasoInicial")
      wire#w2
      S_Coil( "P5" )
   END_RUNG
   RUNG wire#powerrail
      I_Contact( "Datos_Ignition".IGNI_FAC )
      Contact( "Datos_Ignition".AUTO )
   END_RUNG wire#w1
   RUNG wire#w2
      R_Coil( "P4" )
   END_RUNG
   // the same network as SCL:
   #_w1 := (("Datos_Ignition".IGNI_FAC AND "AUTOMATICO") OR (NOT "Datos_Ignition".IGNI_FAC AND "Datos_Ignition".AUTO)) AND "P4" AND NOT "I2_SensorPasoInicial" AND "FN_I2_SensorPasoInicial";   // falling edge of "I2_SensorPasoInicial"
   "FN_I2_SensorPasoInicial" := "I2_SensorPasoInicial";
   IF #_w1 THEN
       "P5" := TRUE;
       "P4" := FALSE;
   END_IF;
END_REGION

REGION Network 7: Lugar P5 => Selector de por color => Blue-Izquierda,Green-> Recto,GreenRugoso-Derecha
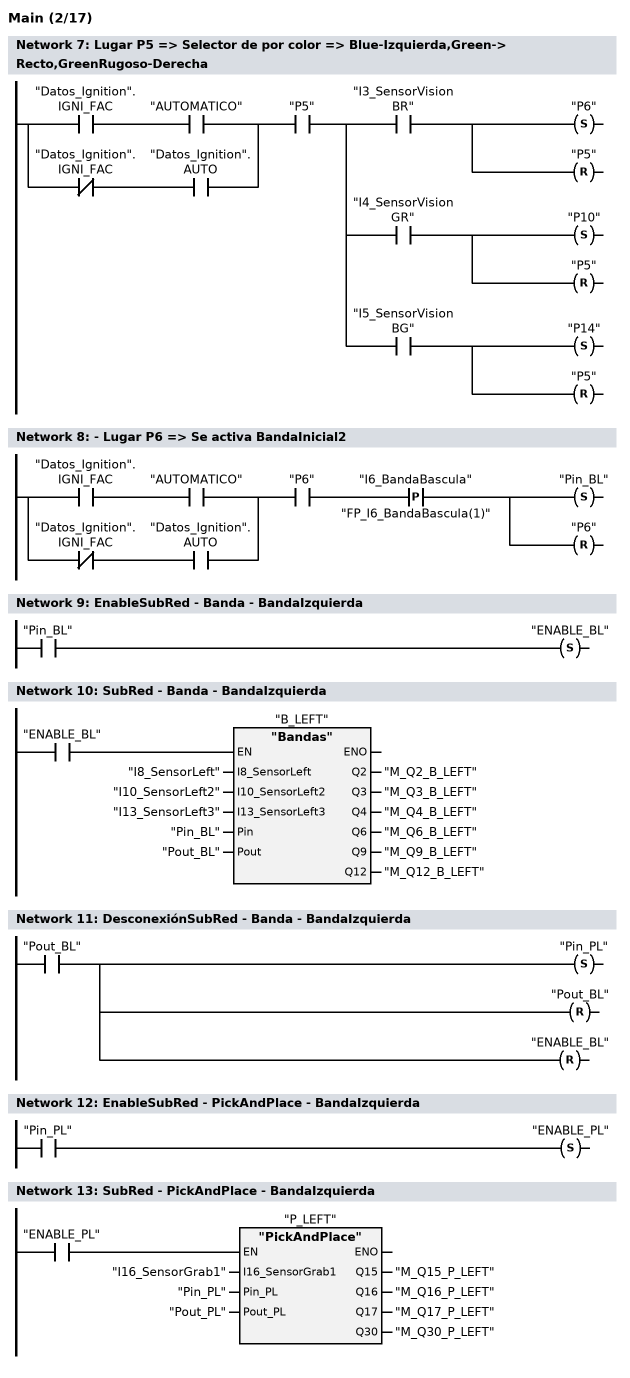
   RUNG wire#powerrail
      Contact( "Datos_Ignition".IGNI_FAC )
      Contact( "AUTOMATICO" )
      wire#w1
      Contact( "P5" )
      wire#w2
      Contact( "I3_SensorVisionBR" )
      wire#w3
      S_Coil( "P6" )
   END_RUNG
   RUNG wire#powerrail
      I_Contact( "Datos_Ignition".IGNI_FAC )
      Contact( "Datos_Ignition".AUTO )
   END_RUNG wire#w1
   RUNG wire#w3
      R_Coil( "P5" )
   END_RUNG
   RUNG wire#w2
      Contact( "I4_SensorVisionGR" )
      wire#w4
      S_Coil( "P10" )
   END_RUNG
   RUNG wire#w4
      R_Coil( "P5" )
   END_RUNG
   RUNG wire#w2
      Contact( "I5_SensorVisionBG" )
      wire#w5
      S_Coil( "P14" )
   END_RUNG
   RUNG wire#w5
      R_Coil( "P5" )
   END_RUNG
   // the same network as SCL:
   #_w1 := (("Datos_Ignition".IGNI_FAC AND "AUTOMATICO") OR (NOT "Datos_Ignition".IGNI_FAC AND "Datos_Ignition".AUTO)) AND "P5";
   IF #_w1 AND "I3_SensorVisionBR" THEN
       "P6" := TRUE;
       "P5" := FALSE;
   END_IF;
   IF #_w1 AND "I4_SensorVisionGR" THEN
       "P10" := TRUE;
       "P5" := FALSE;
   END_IF;
   IF #_w1 AND "I5_SensorVisionBG" THEN
       "P14" := TRUE;
       "P5" := FALSE;
   END_IF;
END_REGION

REGION Network 8: - Lugar P6 => Se activa BandaInicial2
   RUNG wire#powerrail
      Contact( "Datos_Ignition".IGNI_FAC )
      Contact( "AUTOMATICO" )
      wire#w1
      Contact( "P6" )
      P_Contact(operand := "I6_BandaBascula", bit := "FP_I6_BandaBascula(1)")
      wire#w2
      S_Coil( "Pin_BL" )
   END_RUNG
   RUNG wire#powerrail
      I_Contact( "Datos_Ignition".IGNI_FAC )
      Contact( "Datos_Ignition".AUTO )
   END_RUNG wire#w1
   RUNG wire#w2
      R_Coil( "P6" )
   END_RUNG
   // the same network as SCL:
   #_w1 := (("Datos_Ignition".IGNI_FAC AND "AUTOMATICO") OR (NOT "Datos_Ignition".IGNI_FAC AND "Datos_Ignition".AUTO)) AND "P6" AND "I6_BandaBascula" AND NOT "FP_I6_BandaBascula(1)";   // rising edge of "I6_BandaBascula"
   "FP_I6_BandaBascula(1)" := "I6_BandaBascula";
   IF #_w1 THEN
       "Pin_BL" := TRUE;
       "P6" := FALSE;
   END_IF;
END_REGION

REGION Network 9: EnableSubRed - Banda - BandaIzquierda
   RUNG wire#powerrail
      Contact( "Pin_BL" )
      S_Coil( "ENABLE_BL" )
   END_RUNG
   // the same network as SCL:
   IF "Pin_BL" THEN "ENABLE_BL" := TRUE; END_IF;
END_REGION

REGION Network 10: SubRed - Banda - BandaIzquierda
   RUNG wire#powerrail
      Contact( "ENABLE_BL" )
      "B_LEFT"(I8_SensorLeft := "I8_SensorLeft", I10_SensorLeft2 := "I10_SensorLeft2", I13_SensorLeft3 := "I13_SensorLeft3", Pin := "Pin_BL", Pout := "Pout_BL", Q2 => "M_Q2_B_LEFT", Q3 => "M_Q3_B_LEFT", Q4 => "M_Q4_B_LEFT", Q6 => "M_Q6_B_LEFT", Q9 => "M_Q9_B_LEFT", Q12 => "M_Q12_B_LEFT")
   END_RUNG
   // the same network as SCL:
   IF "ENABLE_BL" THEN
       "B_LEFT"(I8_SensorLeft := "I8_SensorLeft",   // "Bandas"
                I10_SensorLeft2 := "I10_SensorLeft2",
                I13_SensorLeft3 := "I13_SensorLeft3",
                Pin := "Pin_BL",
                Pout := "Pout_BL",
                Q2 => "M_Q2_B_LEFT",
                Q3 => "M_Q3_B_LEFT",
                Q4 => "M_Q4_B_LEFT",
                Q6 => "M_Q6_B_LEFT",
                Q9 => "M_Q9_B_LEFT",
                Q12 => "M_Q12_B_LEFT");
   END_IF;
END_REGION

REGION Network 11: DesconexiónSubRed - Banda - BandaIzquierda
   RUNG wire#powerrail
      Contact( "Pout_BL" )
      wire#w1
      S_Coil( "Pin_PL" )
   END_RUNG
   RUNG wire#w1
      R_Coil( "Pout_BL" )
   END_RUNG
   RUNG wire#w1
      R_Coil( "ENABLE_BL" )
   END_RUNG
   // the same network as SCL:
   IF "Pout_BL" THEN "Pin_PL" := TRUE; END_IF;
   #_w1 := "Pout_BL";
   IF #_w1 THEN
       "Pout_BL" := FALSE;
       "ENABLE_BL" := FALSE;
   END_IF;
END_REGION

REGION Network 12: EnableSubRed - PickAndPlace - BandaIzquierda
   RUNG wire#powerrail
      Contact( "Pin_PL" )
      S_Coil( "ENABLE_PL" )
   END_RUNG
   // the same network as SCL:
   IF "Pin_PL" THEN "ENABLE_PL" := TRUE; END_IF;
END_REGION

REGION Network 13: SubRed - PickAndPlace - BandaIzquierda
   RUNG wire#powerrail
      Contact( "ENABLE_PL" )
      "P_LEFT"(I16_SensorGrab1 := "I16_SensorGrab1", Pin_PL := "Pin_PL", Pout_PL := "Pout_PL", Q15 => "M_Q15_P_LEFT", Q16 => "M_Q16_P_LEFT", Q17 => "M_Q17_P_LEFT", Q30 => "M_Q30_P_LEFT")
   END_RUNG
   // the same network as SCL:
   IF "ENABLE_PL" THEN
       "P_LEFT"(I16_SensorGrab1 := "I16_SensorGrab1",   // "PickAndPlace"
                Pin_PL := "Pin_PL",
                Pout_PL := "Pout_PL",
                Q15 => "M_Q15_P_LEFT",
                Q16 => "M_Q16_P_LEFT",
                Q17 => "M_Q17_P_LEFT",
                Q30 => "M_Q30_P_LEFT");
   END_IF;
END_REGION

REGION Network 14: DesconexiónSubRed - PickAndPlace - BandaIzquierda
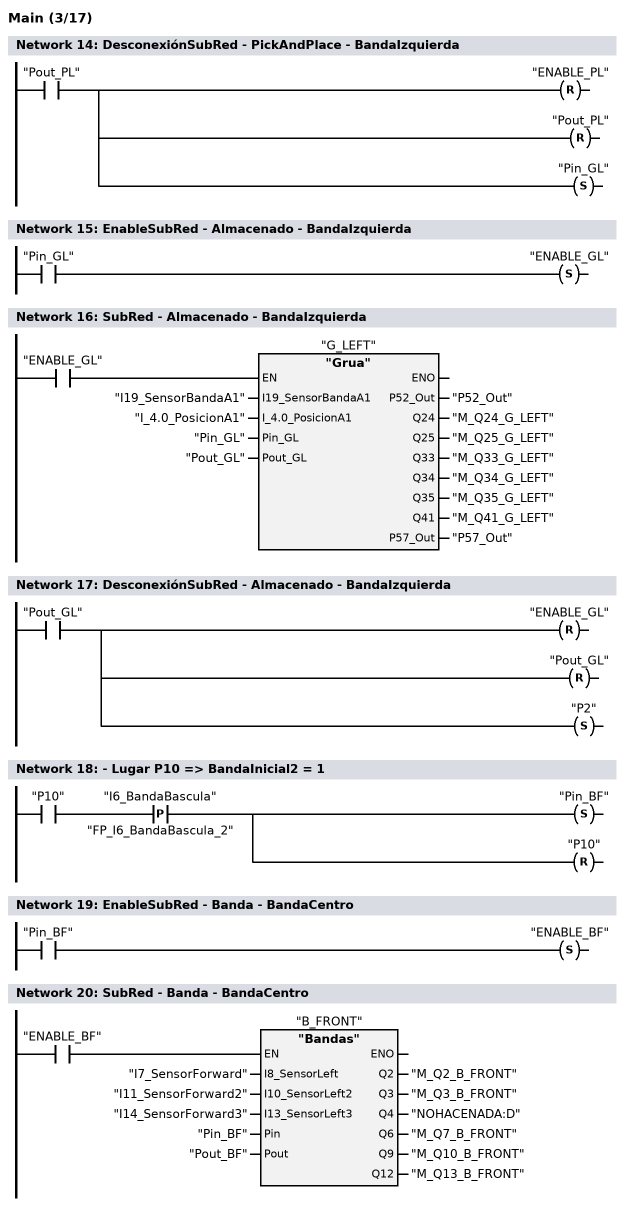
   RUNG wire#powerrail
      Contact( "Pout_PL" )
      wire#w1
      R_Coil( "ENABLE_PL" )
   END_RUNG
   RUNG wire#w1
      R_Coil( "Pout_PL" )
   END_RUNG
   RUNG wire#w1
      S_Coil( "Pin_GL" )
   END_RUNG
   // the same network as SCL:
   IF "Pout_PL" THEN "ENABLE_PL" := FALSE; END_IF;
   #_w1 := "Pout_PL";
   IF #_w1 THEN
       "Pout_PL" := FALSE;
       "Pin_GL" := TRUE;
   END_IF;
END_REGION

REGION Network 15: EnableSubRed - Almacenado - BandaIzquierda
   RUNG wire#powerrail
      Contact( "Pin_GL" )
      S_Coil( "ENABLE_GL" )
   END_RUNG
   // the same network as SCL:
   IF "Pin_GL" THEN "ENABLE_GL" := TRUE; END_IF;
END_REGION

REGION Network 16: SubRed - Almacenado - BandaIzquierda
   RUNG wire#powerrail
      Contact( "ENABLE_GL" )
      "G_LEFT"(I19_SensorBandaA1 := "I19_SensorBandaA1", "I_4.0_PosicionA1" := "I_4.0_PosicionA1", Pin_GL := "Pin_GL", Pout_GL := "Pout_GL", P52_Out => "P52_Out", Q24 => "M_Q24_G_LEFT", Q25 => "M_Q25_G_LEFT", Q33 => "M_Q33_G_LEFT", Q34 => "M_Q34_G_LEFT", Q35 => "M_Q35_G_LEFT", Q41 => "M_Q41_G_LEFT", P57_Out => "P57_Out")
   END_RUNG
   // the same network as SCL:
   IF "ENABLE_GL" THEN
       "G_LEFT"(I19_SensorBandaA1 := "I19_SensorBandaA1",   // "Grua"
                "I_4.0_PosicionA1" := "I_4.0_PosicionA1",
                Pin_GL := "Pin_GL",
                Pout_GL := "Pout_GL",
                P52_Out => "P52_Out",
                Q24 => "M_Q24_G_LEFT",
                Q25 => "M_Q25_G_LEFT",
                Q33 => "M_Q33_G_LEFT",
                Q34 => "M_Q34_G_LEFT",
                Q35 => "M_Q35_G_LEFT",
                Q41 => "M_Q41_G_LEFT",
                P57_Out => "P57_Out");
   END_IF;
END_REGION

REGION Network 17: DesconexiónSubRed - Almacenado - BandaIzquierda
   RUNG wire#powerrail
      Contact( "Pout_GL" )
      wire#w1
      R_Coil( "ENABLE_GL" )
   END_RUNG
   RUNG wire#w1
      R_Coil( "Pout_GL" )
   END_RUNG
   RUNG wire#w1
      S_Coil( "P2" )
   END_RUNG
   // the same network as SCL:
   IF "Pout_GL" THEN "ENABLE_GL" := FALSE; END_IF;
   #_w1 := "Pout_GL";
   IF #_w1 THEN
       "Pout_GL" := FALSE;
       "P2" := TRUE;
   END_IF;
END_REGION

REGION Network 18: - Lugar P10 => BandaInicial2 = 1
   RUNG wire#powerrail
      Contact( "P10" )
      P_Contact(operand := "I6_BandaBascula", bit := "FP_I6_BandaBascula_2")
      wire#w1
      S_Coil( "Pin_BF" )
   END_RUNG
   RUNG wire#w1
      R_Coil( "P10" )
   END_RUNG
   // the same network as SCL:
   #_w1 := "P10" AND "I6_BandaBascula" AND NOT "FP_I6_BandaBascula_2";   // rising edge of "I6_BandaBascula"
   "FP_I6_BandaBascula_2" := "I6_BandaBascula";
   IF #_w1 THEN
       "Pin_BF" := TRUE;
       "P10" := FALSE;
   END_IF;
END_REGION

REGION Network 19: EnableSubRed - Banda - BandaCentro
   RUNG wire#powerrail
      Contact( "Pin_BF" )
      S_Coil( "ENABLE_BF" )
   END_RUNG
   // the same network as SCL:
   IF "Pin_BF" THEN "ENABLE_BF" := TRUE; END_IF;
END_REGION

REGION Network 20: SubRed - Banda - BandaCentro
   RUNG wire#powerrail
      Contact( "ENABLE_BF" )
      "B_FRONT"(I8_SensorLeft := "I7_SensorForward", I10_SensorLeft2 := "I11_SensorForward2", I13_SensorLeft3 := "I14_SensorForward3", Pin := "Pin_BF", Pout := "Pout_BF", Q2 => "M_Q2_B_FRONT", Q3 => "M_Q3_B_FRONT", Q4 => "NOHACENADA:D", Q6 => "M_Q7_B_FRONT", Q9 => "M_Q10_B_FRONT", Q12 => "M_Q13_B_FRONT")
   END_RUNG
   // the same network as SCL:
   IF "ENABLE_BF" THEN
       "B_FRONT"(I8_SensorLeft := "I7_SensorForward",   // "Bandas"
                 I10_SensorLeft2 := "I11_SensorForward2",
                 I13_SensorLeft3 := "I14_SensorForward3",
                 Pin := "Pin_BF",
                 Pout := "Pout_BF",
                 Q2 => "M_Q2_B_FRONT",
                 Q3 => "M_Q3_B_FRONT",
                 Q4 => "NOHACENADA:D",
                 Q6 => "M_Q7_B_FRONT",
                 Q9 => "M_Q10_B_FRONT",
                 Q12 => "M_Q13_B_FRONT");
   END_IF;
END_REGION

REGION Network 21: DesconexiónSubRed - Banda - BandaCentro
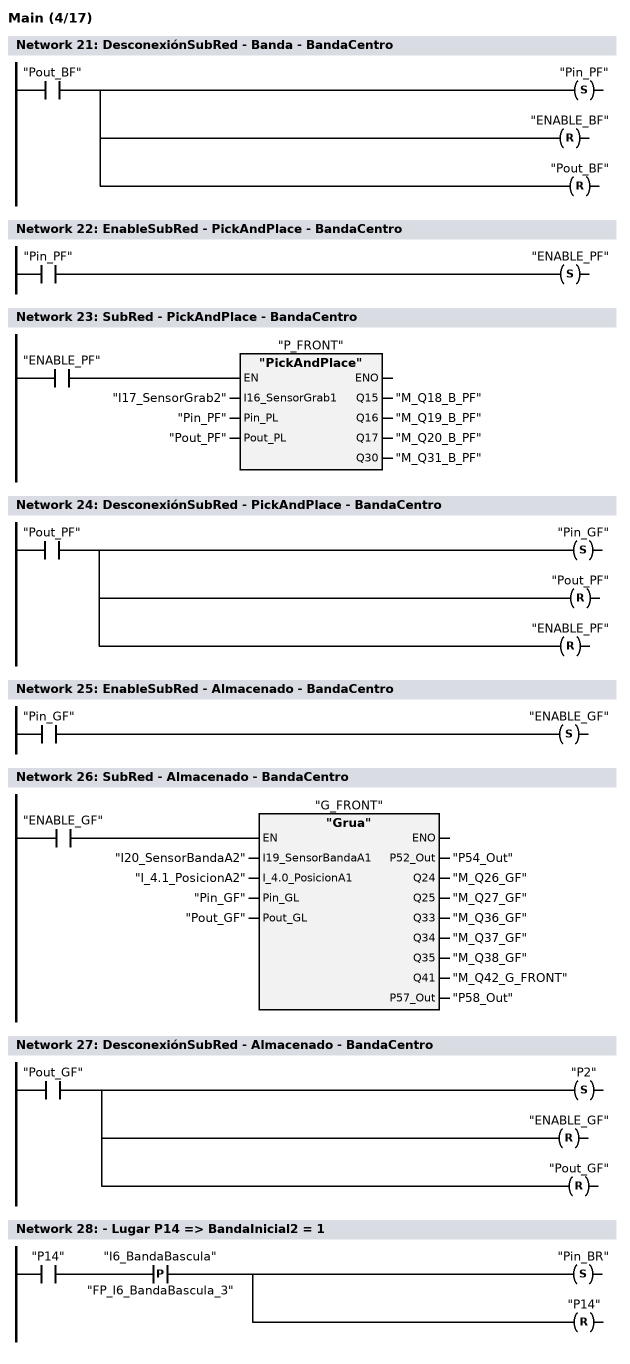
   RUNG wire#powerrail
      Contact( "Pout_BF" )
      wire#w1
      S_Coil( "Pin_PF" )
   END_RUNG
   RUNG wire#w1
      R_Coil( "ENABLE_BF" )
   END_RUNG
   RUNG wire#w1
      R_Coil( "Pout_BF" )
   END_RUNG
   // the same network as SCL:
   IF "Pout_BF" THEN
       "Pin_PF" := TRUE;
       "ENABLE_BF" := FALSE;
       "Pout_BF" := FALSE;
   END_IF;
END_REGION

REGION Network 22: EnableSubRed - PickAndPlace - BandaCentro
   RUNG wire#powerrail
      Contact( "Pin_PF" )
      S_Coil( "ENABLE_PF" )
   END_RUNG
   // the same network as SCL:
   IF "Pin_PF" THEN "ENABLE_PF" := TRUE; END_IF;
END_REGION

REGION Network 23: SubRed - PickAndPlace - BandaCentro
   RUNG wire#powerrail
      Contact( "ENABLE_PF" )
      "P_FRONT"(I16_SensorGrab1 := "I17_SensorGrab2", Pin_PL := "Pin_PF", Pout_PL := "Pout_PF", Q15 => "M_Q18_B_PF", Q16 => "M_Q19_B_PF", Q17 => "M_Q20_B_PF", Q30 => "M_Q31_B_PF")
   END_RUNG
   // the same network as SCL:
   IF "ENABLE_PF" THEN
       "P_FRONT"(I16_SensorGrab1 := "I17_SensorGrab2",   // "PickAndPlace"
                 Pin_PL := "Pin_PF",
                 Pout_PL := "Pout_PF",
                 Q15 => "M_Q18_B_PF",
                 Q16 => "M_Q19_B_PF",
                 Q17 => "M_Q20_B_PF",
                 Q30 => "M_Q31_B_PF");
   END_IF;
END_REGION

REGION Network 24: DesconexiónSubRed - PickAndPlace - BandaCentro
   RUNG wire#powerrail
      Contact( "Pout_PF" )
      wire#w1
      S_Coil( "Pin_GF" )
   END_RUNG
   RUNG wire#w1
      R_Coil( "Pout_PF" )
   END_RUNG
   RUNG wire#w1
      R_Coil( "ENABLE_PF" )
   END_RUNG
   // the same network as SCL:
   IF "Pout_PF" THEN "Pin_GF" := TRUE; END_IF;
   #_w1 := "Pout_PF";
   IF #_w1 THEN
       "Pout_PF" := FALSE;
       "ENABLE_PF" := FALSE;
   END_IF;
END_REGION

REGION Network 25: EnableSubRed - Almacenado - BandaCentro
   RUNG wire#powerrail
      Contact( "Pin_GF" )
      S_Coil( "ENABLE_GF" )
   END_RUNG
   // the same network as SCL:
   IF "Pin_GF" THEN "ENABLE_GF" := TRUE; END_IF;
END_REGION

REGION Network 26: SubRed - Almacenado - BandaCentro
   RUNG wire#powerrail
      Contact( "ENABLE_GF" )
      "G_FRONT"(I19_SensorBandaA1 := "I20_SensorBandaA2", "I_4.0_PosicionA1" := "I_4.1_PosicionA2", Pin_GL := "Pin_GF", Pout_GL := "Pout_GF", P52_Out => "P54_Out", Q24 => "M_Q26_GF", Q25 => "M_Q27_GF", Q33 => "M_Q36_GF", Q34 => "M_Q37_GF", Q35 => "M_Q38_GF", Q41 => "M_Q42_G_FRONT", P57_Out => "P58_Out")
   END_RUNG
   // the same network as SCL:
   IF "ENABLE_GF" THEN
       "G_FRONT"(I19_SensorBandaA1 := "I20_SensorBandaA2",   // "Grua"
                 "I_4.0_PosicionA1" := "I_4.1_PosicionA2",
                 Pin_GL := "Pin_GF",
                 Pout_GL := "Pout_GF",
                 P52_Out => "P54_Out",
                 Q24 => "M_Q26_GF",
                 Q25 => "M_Q27_GF",
                 Q33 => "M_Q36_GF",
                 Q34 => "M_Q37_GF",
                 Q35 => "M_Q38_GF",
                 Q41 => "M_Q42_G_FRONT",
                 P57_Out => "P58_Out");
   END_IF;
END_REGION

REGION Network 27: DesconexiónSubRed - Almacenado - BandaCentro
   RUNG wire#powerrail
      Contact( "Pout_GF" )
      wire#w1
      S_Coil( "P2" )
   END_RUNG
   RUNG wire#w1
      R_Coil( "ENABLE_GF" )
   END_RUNG
   RUNG wire#w1
      R_Coil( "Pout_GF" )
   END_RUNG
   // the same network as SCL:
   IF "Pout_GF" THEN
       "P2" := TRUE;
       "ENABLE_GF" := FALSE;
       "Pout_GF" := FALSE;
   END_IF;
END_REGION

REGION Network 28: - Lugar P14 => BandaInicial2 = 1
   RUNG wire#powerrail
      Contact( "P14" )
      P_Contact(operand := "I6_BandaBascula", bit := "FP_I6_BandaBascula_3")
      wire#w1
      S_Coil( "Pin_BR" )
   END_RUNG
   RUNG wire#w1
      R_Coil( "P14" )
   END_RUNG
   // the same network as SCL:
   #_w1 := "P14" AND "I6_BandaBascula" AND NOT "FP_I6_BandaBascula_3";   // rising edge of "I6_BandaBascula"
   "FP_I6_BandaBascula_3" := "I6_BandaBascula";
   IF #_w1 THEN
       "Pin_BR" := TRUE;
       "P14" := FALSE;
   END_IF;
END_REGION

REGION Network 29: EnableSubRed - Banda - BandaDerecha
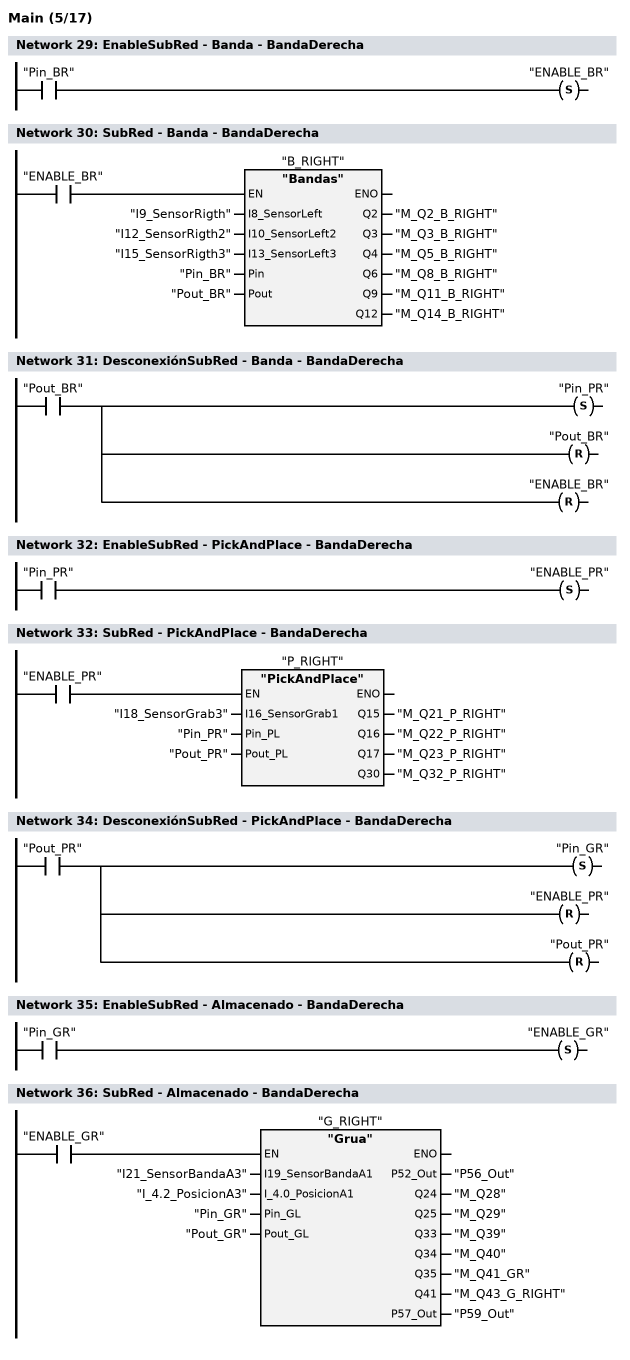
   RUNG wire#powerrail
      Contact( "Pin_BR" )
      S_Coil( "ENABLE_BR" )
   END_RUNG
   // the same network as SCL:
   IF "Pin_BR" THEN "ENABLE_BR" := TRUE; END_IF;
END_REGION

REGION Network 30: SubRed - Banda - BandaDerecha
   RUNG wire#powerrail
      Contact( "ENABLE_BR" )
      "B_RIGHT"(I8_SensorLeft := "I9_SensorRigth", I10_SensorLeft2 := "I12_SensorRigth2", I13_SensorLeft3 := "I15_SensorRigth3", Pin := "Pin_BR", Pout := "Pout_BR", Q2 => "M_Q2_B_RIGHT", Q3 => "M_Q3_B_RIGHT", Q4 => "M_Q5_B_RIGHT", Q6 => "M_Q8_B_RIGHT", Q9 => "M_Q11_B_RIGHT", Q12 => "M_Q14_B_RIGHT")
   END_RUNG
   // the same network as SCL:
   IF "ENABLE_BR" THEN
       "B_RIGHT"(I8_SensorLeft := "I9_SensorRigth",   // "Bandas"
                 I10_SensorLeft2 := "I12_SensorRigth2",
                 I13_SensorLeft3 := "I15_SensorRigth3",
                 Pin := "Pin_BR",
                 Pout := "Pout_BR",
                 Q2 => "M_Q2_B_RIGHT",
                 Q3 => "M_Q3_B_RIGHT",
                 Q4 => "M_Q5_B_RIGHT",
                 Q6 => "M_Q8_B_RIGHT",
                 Q9 => "M_Q11_B_RIGHT",
                 Q12 => "M_Q14_B_RIGHT");
   END_IF;
END_REGION

REGION Network 31: DesconexiónSubRed - Banda - BandaDerecha
   RUNG wire#powerrail
      Contact( "Pout_BR" )
      wire#w1
      S_Coil( "Pin_PR" )
   END_RUNG
   RUNG wire#w1
      R_Coil( "Pout_BR" )
   END_RUNG
   RUNG wire#w1
      R_Coil( "ENABLE_BR" )
   END_RUNG
   // the same network as SCL:
   IF "Pout_BR" THEN "Pin_PR" := TRUE; END_IF;
   #_w1 := "Pout_BR";
   IF #_w1 THEN
       "Pout_BR" := FALSE;
       "ENABLE_BR" := FALSE;
   END_IF;
END_REGION

REGION Network 32: EnableSubRed - PickAndPlace - BandaDerecha
   RUNG wire#powerrail
      Contact( "Pin_PR" )
      S_Coil( "ENABLE_PR" )
   END_RUNG
   // the same network as SCL:
   IF "Pin_PR" THEN "ENABLE_PR" := TRUE; END_IF;
END_REGION

REGION Network 33: SubRed - PickAndPlace - BandaDerecha
   RUNG wire#powerrail
      Contact( "ENABLE_PR" )
      "P_RIGHT"(I16_SensorGrab1 := "I18_SensorGrab3", Pin_PL := "Pin_PR", Pout_PL := "Pout_PR", Q15 => "M_Q21_P_RIGHT", Q16 => "M_Q22_P_RIGHT", Q17 => "M_Q23_P_RIGHT", Q30 => "M_Q32_P_RIGHT")
   END_RUNG
   // the same network as SCL:
   IF "ENABLE_PR" THEN
       "P_RIGHT"(I16_SensorGrab1 := "I18_SensorGrab3",   // "PickAndPlace"
                 Pin_PL := "Pin_PR",
                 Pout_PL := "Pout_PR",
                 Q15 => "M_Q21_P_RIGHT",
                 Q16 => "M_Q22_P_RIGHT",
                 Q17 => "M_Q23_P_RIGHT",
                 Q30 => "M_Q32_P_RIGHT");
   END_IF;
END_REGION

REGION Network 34: DesconexiónSubRed - PickAndPlace - BandaDerecha
   RUNG wire#powerrail
      Contact( "Pout_PR" )
      wire#w1
      S_Coil( "Pin_GR" )
   END_RUNG
   RUNG wire#w1
      R_Coil( "ENABLE_PR" )
   END_RUNG
   RUNG wire#w1
      R_Coil( "Pout_PR" )
   END_RUNG
   // the same network as SCL:
   IF "Pout_PR" THEN
       "Pin_GR" := TRUE;
       "ENABLE_PR" := FALSE;
       "Pout_PR" := FALSE;
   END_IF;
END_REGION

REGION Network 35: EnableSubRed - Almacenado - BandaDerecha
   RUNG wire#powerrail
      Contact( "Pin_GR" )
      S_Coil( "ENABLE_GR" )
   END_RUNG
   // the same network as SCL:
   IF "Pin_GR" THEN "ENABLE_GR" := TRUE; END_IF;
END_REGION

REGION Network 36: SubRed - Almacenado - BandaDerecha
   RUNG wire#powerrail
      Contact( "ENABLE_GR" )
      "G_RIGHT"(I19_SensorBandaA1 := "I21_SensorBandaA3", "I_4.0_PosicionA1" := "I_4.2_PosicionA3", Pin_GL := "Pin_GR", Pout_GL := "Pout_GR", P52_Out => "P56_Out", Q24 => "M_Q28", Q25 => "M_Q29", Q33 => "M_Q39", Q34 => "M_Q40", Q35 => "M_Q41_GR", Q41 => "M_Q43_G_RIGHT", P57_Out => "P59_Out")
   END_RUNG
   // the same network as SCL:
   IF "ENABLE_GR" THEN
       "G_RIGHT"(I19_SensorBandaA1 := "I21_SensorBandaA3",   // "Grua"
                 "I_4.0_PosicionA1" := "I_4.2_PosicionA3",
                 Pin_GL := "Pin_GR",
                 Pout_GL := "Pout_GR",
                 P52_Out => "P56_Out",
                 Q24 => "M_Q28",
                 Q25 => "M_Q29",
                 Q33 => "M_Q39",
                 Q34 => "M_Q40",
                 Q35 => "M_Q41_GR",
                 Q41 => "M_Q43_G_RIGHT",
                 P57_Out => "P59_Out");
   END_IF;
END_REGION

REGION Network 37: DesconexiónSubRed - Almacenado - BandaDerecha
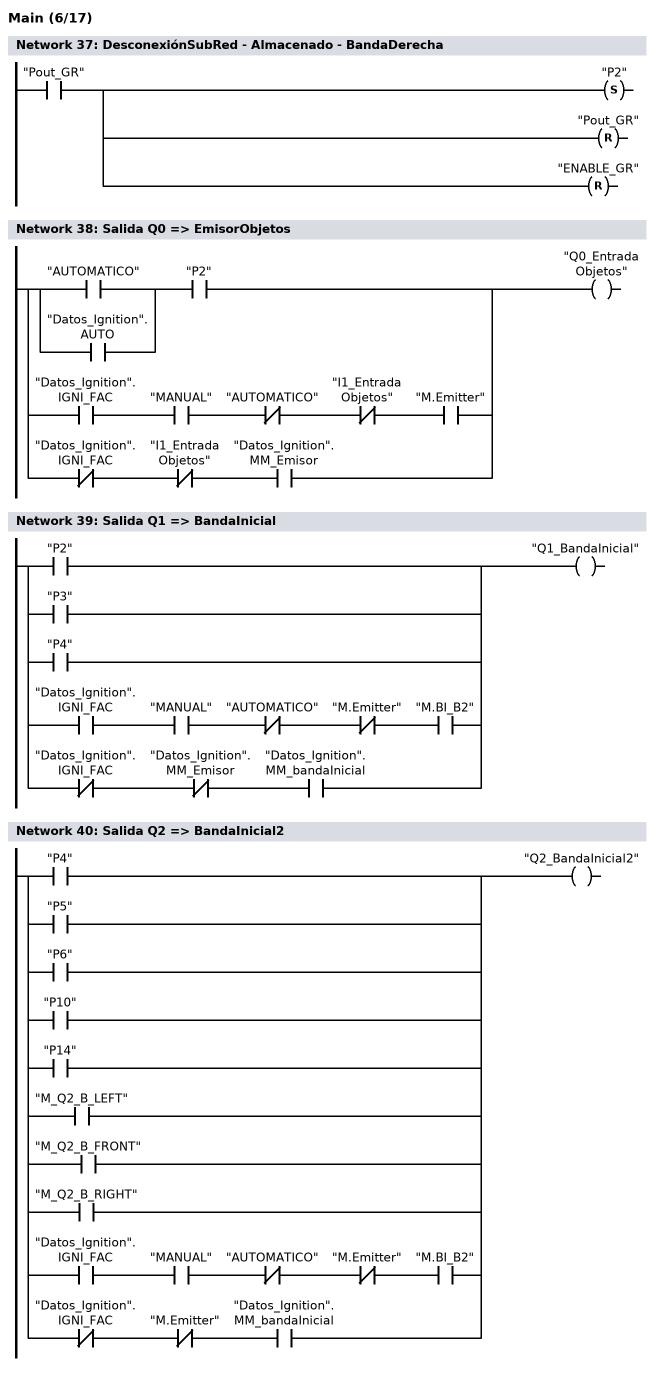
   RUNG wire#powerrail
      Contact( "Pout_GR" )
      wire#w1
      S_Coil( "P2" )
   END_RUNG
   RUNG wire#w1
      R_Coil( "Pout_GR" )
   END_RUNG
   RUNG wire#w1
      R_Coil( "ENABLE_GR" )
   END_RUNG
   // the same network as SCL:
   IF "Pout_GR" THEN "P2" := TRUE; END_IF;
   #_w1 := "Pout_GR";
   IF #_w1 THEN
       "Pout_GR" := FALSE;
       "ENABLE_GR" := FALSE;
   END_IF;
END_REGION

REGION Network 38: Salida Q0 => EmisorObjetos
   RUNG wire#powerrail
      Contact( "AUTOMATICO" )
      wire#w1
      Contact( "P2" )
      wire#w2
      Coil( "Q0_EntradaObjetos" )
   END_RUNG
   RUNG wire#powerrail
      Contact( "Datos_Ignition".AUTO )
   END_RUNG wire#w1
   RUNG wire#powerrail
      Contact( "Datos_Ignition".IGNI_FAC )
      Contact( "MANUAL" )
      I_Contact( "AUTOMATICO" )
      I_Contact( "I1_EntradaObjetos" )
      Contact( "M.Emitter" )
   END_RUNG wire#w2
   RUNG wire#powerrail
      I_Contact( "Datos_Ignition".IGNI_FAC )
      I_Contact( "I1_EntradaObjetos" )
      Contact( "Datos_Ignition".MM_Emisor )
   END_RUNG wire#w2
   // the same network as SCL:
   "Q0_EntradaObjetos" := (("AUTOMATICO" OR "Datos_Ignition".AUTO) AND "P2") OR ("Datos_Ignition".IGNI_FAC AND "MANUAL" AND NOT "AUTOMATICO" AND NOT "I1_EntradaObjetos" AND "M.Emitter") OR (NOT "Datos_Ignition".IGNI_FAC AND NOT "I1_EntradaObjetos" AND "Datos_Ignition".MM_Emisor);
END_REGION

REGION Network 39: Salida Q1 => BandaInicial
   RUNG wire#powerrail
      Contact( "P2" )
      wire#w1
      Coil( "Q1_BandaInicial" )
   END_RUNG
   RUNG wire#powerrail
      Contact( "P3" )
   END_RUNG wire#w1
   RUNG wire#powerrail
      Contact( "P4" )
   END_RUNG wire#w1
   RUNG wire#powerrail
      Contact( "Datos_Ignition".IGNI_FAC )
      Contact( "MANUAL" )
      I_Contact( "AUTOMATICO" )
      I_Contact( "M.Emitter" )
      Contact( "M.BI_B2" )
   END_RUNG wire#w1
   RUNG wire#powerrail
      I_Contact( "Datos_Ignition".IGNI_FAC )
      I_Contact( "Datos_Ignition".MM_Emisor )
      Contact( "Datos_Ignition".MM_bandaInicial )
   END_RUNG wire#w1
   // the same network as SCL:
   "Q1_BandaInicial" := "P2" OR "P3" OR "P4" OR ("Datos_Ignition".IGNI_FAC AND "MANUAL" AND NOT "AUTOMATICO" AND NOT "M.Emitter" AND "M.BI_B2") OR (NOT "Datos_Ignition".IGNI_FAC AND NOT "Datos_Ignition".MM_Emisor AND "Datos_Ignition".MM_bandaInicial);
END_REGION

REGION Network 40: Salida Q2 => BandaInicial2
   RUNG wire#powerrail
      Contact( "P4" )
      wire#w1
      Coil( "Q2_BandaInicial2" )
   END_RUNG
   RUNG wire#powerrail
      Contact( "P5" )
   END_RUNG wire#w1
   RUNG wire#powerrail
      Contact( "P6" )
   END_RUNG wire#w1
   RUNG wire#powerrail
      Contact( "P10" )
   END_RUNG wire#w1
   RUNG wire#powerrail
      Contact( "P14" )
   END_RUNG wire#w1
   RUNG wire#powerrail
      Contact( "M_Q2_B_LEFT" )
   END_RUNG wire#w1
   RUNG wire#powerrail
      Contact( "M_Q2_B_FRONT" )
   END_RUNG wire#w1
   RUNG wire#powerrail
      Contact( "M_Q2_B_RIGHT" )
   END_RUNG wire#w1
   RUNG wire#powerrail
      Contact( "Datos_Ignition".IGNI_FAC )
      Contact( "MANUAL" )
      I_Contact( "AUTOMATICO" )
      I_Contact( "M.Emitter" )
      Contact( "M.BI_B2" )
   END_RUNG wire#w1
   RUNG wire#powerrail
      I_Contact( "Datos_Ignition".IGNI_FAC )
      I_Contact( "M.Emitter" )
      Contact( "Datos_Ignition".MM_bandaInicial )
   END_RUNG wire#w1
   // the same network as SCL:
   "Q2_BandaInicial2" := "P4" OR "P5" OR "P6" OR "P10" OR "P14" OR "M_Q2_B_LEFT" OR "M_Q2_B_FRONT" OR "M_Q2_B_RIGHT" OR ("Datos_Ignition".IGNI_FAC AND "MANUAL" AND NOT "AUTOMATICO" AND NOT "M.Emitter" AND "M.BI_B2") OR (NOT "Datos_Ignition".IGNI_FAC AND NOT "M.Emitter" AND "Datos_Ignition".MM_bandaInicial);
END_REGION

REGION Network 41: Salida Q3 => RuedasForward
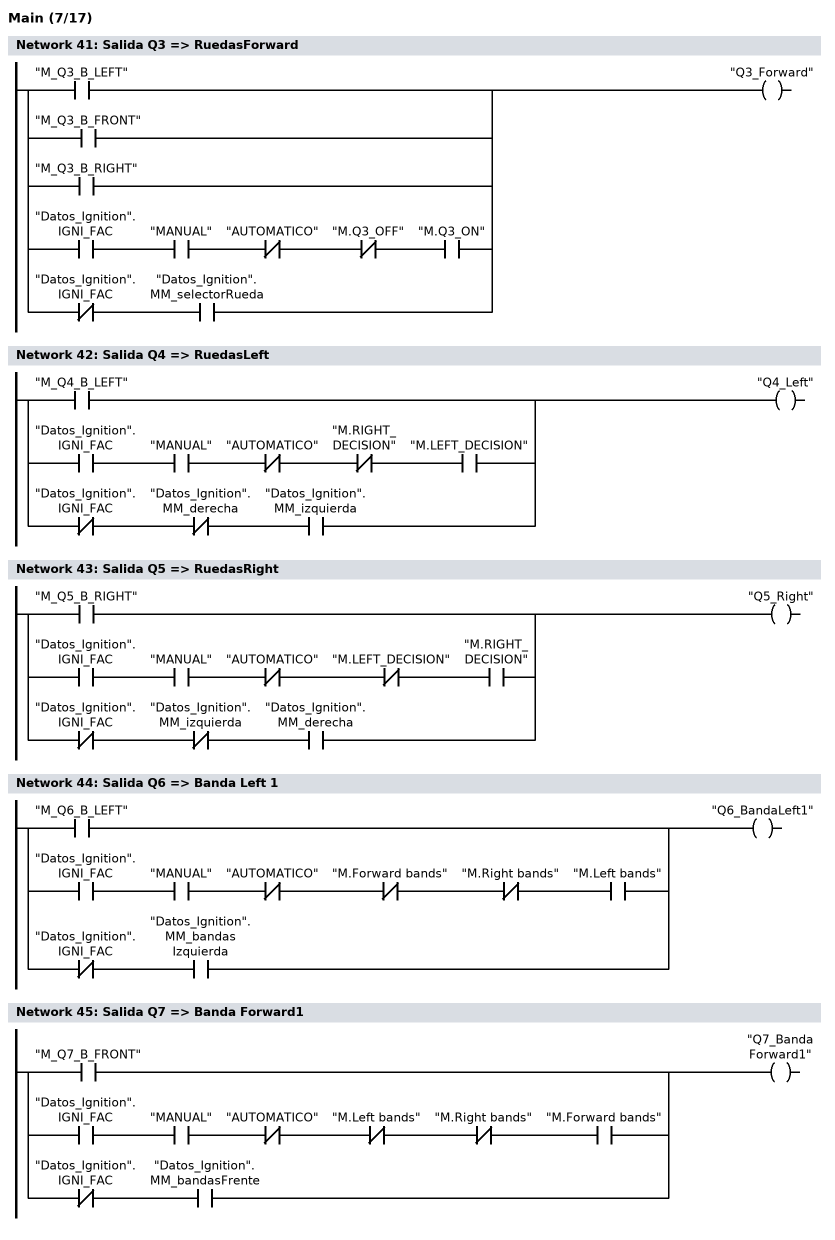
   RUNG wire#powerrail
      Contact( "M_Q3_B_LEFT" )
      wire#w1
      Coil( "Q3_Forward" )
   END_RUNG
   RUNG wire#powerrail
      Contact( "M_Q3_B_FRONT" )
   END_RUNG wire#w1
   RUNG wire#powerrail
      Contact( "M_Q3_B_RIGHT" )
   END_RUNG wire#w1
   RUNG wire#powerrail
      Contact( "Datos_Ignition".IGNI_FAC )
      Contact( "MANUAL" )
      I_Contact( "AUTOMATICO" )
      I_Contact( "M.Q3_OFF" )
      Contact( "M.Q3_ON" )
   END_RUNG wire#w1
   RUNG wire#powerrail
      I_Contact( "Datos_Ignition".IGNI_FAC )
      Contact( "Datos_Ignition".MM_selectorRueda )
   END_RUNG wire#w1
   // the same network as SCL:
   "Q3_Forward" := "M_Q3_B_LEFT" OR "M_Q3_B_FRONT" OR "M_Q3_B_RIGHT" OR ("Datos_Ignition".IGNI_FAC AND "MANUAL" AND NOT "AUTOMATICO" AND NOT "M.Q3_OFF" AND "M.Q3_ON") OR (NOT "Datos_Ignition".IGNI_FAC AND "Datos_Ignition".MM_selectorRueda);
END_REGION

REGION Network 42: Salida Q4 => RuedasLeft
   RUNG wire#powerrail
      Contact( "M_Q4_B_LEFT" )
      wire#w1
      Coil( "Q4_Left" )
   END_RUNG
   RUNG wire#powerrail
      Contact( "Datos_Ignition".IGNI_FAC )
      Contact( "MANUAL" )
      I_Contact( "AUTOMATICO" )
      I_Contact( "M.RIGHT_DECISION" )
      Contact( "M.LEFT_DECISION" )
   END_RUNG wire#w1
   RUNG wire#powerrail
      I_Contact( "Datos_Ignition".IGNI_FAC )
      I_Contact( "Datos_Ignition".MM_derecha )
      Contact( "Datos_Ignition".MM_izquierda )
   END_RUNG wire#w1
   // the same network as SCL:
   "Q4_Left" := "M_Q4_B_LEFT" OR ("Datos_Ignition".IGNI_FAC AND "MANUAL" AND NOT "AUTOMATICO" AND NOT "M.RIGHT_DECISION" AND "M.LEFT_DECISION") OR (NOT "Datos_Ignition".IGNI_FAC AND NOT "Datos_Ignition".MM_derecha AND "Datos_Ignition".MM_izquierda);
END_REGION

REGION Network 43: Salida Q5 => RuedasRight
   RUNG wire#powerrail
      Contact( "M_Q5_B_RIGHT" )
      wire#w1
      Coil( "Q5_Right" )
   END_RUNG
   RUNG wire#powerrail
      Contact( "Datos_Ignition".IGNI_FAC )
      Contact( "MANUAL" )
      I_Contact( "AUTOMATICO" )
      I_Contact( "M.LEFT_DECISION" )
      Contact( "M.RIGHT_DECISION" )
   END_RUNG wire#w1
   RUNG wire#powerrail
      I_Contact( "Datos_Ignition".IGNI_FAC )
      I_Contact( "Datos_Ignition".MM_izquierda )
      Contact( "Datos_Ignition".MM_derecha )
   END_RUNG wire#w1
   // the same network as SCL:
   "Q5_Right" := "M_Q5_B_RIGHT" OR ("Datos_Ignition".IGNI_FAC AND "MANUAL" AND NOT "AUTOMATICO" AND NOT "M.LEFT_DECISION" AND "M.RIGHT_DECISION") OR (NOT "Datos_Ignition".IGNI_FAC AND NOT "Datos_Ignition".MM_izquierda AND "Datos_Ignition".MM_derecha);
END_REGION

REGION Network 44: Salida Q6 => Banda Left 1
   RUNG wire#powerrail
      Contact( "M_Q6_B_LEFT" )
      wire#w1
      Coil( "Q6_BandaLeft1" )
   END_RUNG
   RUNG wire#powerrail
      Contact( "Datos_Ignition".IGNI_FAC )
      Contact( "MANUAL" )
      I_Contact( "AUTOMATICO" )
      I_Contact( "M.Forward bands" )
      I_Contact( "M.Right bands" )
      Contact( "M.Left bands" )
   END_RUNG wire#w1
   RUNG wire#powerrail
      I_Contact( "Datos_Ignition".IGNI_FAC )
      Contact( "Datos_Ignition".MM_bandasIzquierda )
   END_RUNG wire#w1
   // the same network as SCL:
   "Q6_BandaLeft1" := "M_Q6_B_LEFT" OR ("Datos_Ignition".IGNI_FAC AND "MANUAL" AND NOT "AUTOMATICO" AND NOT "M.Forward bands" AND NOT "M.Right bands" AND "M.Left bands") OR (NOT "Datos_Ignition".IGNI_FAC AND "Datos_Ignition".MM_bandasIzquierda);
END_REGION

REGION Network 45: Salida Q7 => Banda Forward1
   RUNG wire#powerrail
      Contact( "M_Q7_B_FRONT" )
      wire#w1
      Coil( "Q7_BandaForward1" )
   END_RUNG
   RUNG wire#powerrail
      Contact( "Datos_Ignition".IGNI_FAC )
      Contact( "MANUAL" )
      I_Contact( "AUTOMATICO" )
      I_Contact( "M.Left bands" )
      I_Contact( "M.Right bands" )
      Contact( "M.Forward bands" )
   END_RUNG wire#w1
   RUNG wire#powerrail
      I_Contact( "Datos_Ignition".IGNI_FAC )
      Contact( "Datos_Ignition".MM_bandasFrente )
   END_RUNG wire#w1
   // the same network as SCL:
   "Q7_BandaForward1" := "M_Q7_B_FRONT" OR ("Datos_Ignition".IGNI_FAC AND "MANUAL" AND NOT "AUTOMATICO" AND NOT "M.Left bands" AND NOT "M.Right bands" AND "M.Forward bands") OR (NOT "Datos_Ignition".IGNI_FAC AND "Datos_Ignition".MM_bandasFrente);
END_REGION

REGION Network 46: Salida Q8 => Banda Rigth 1
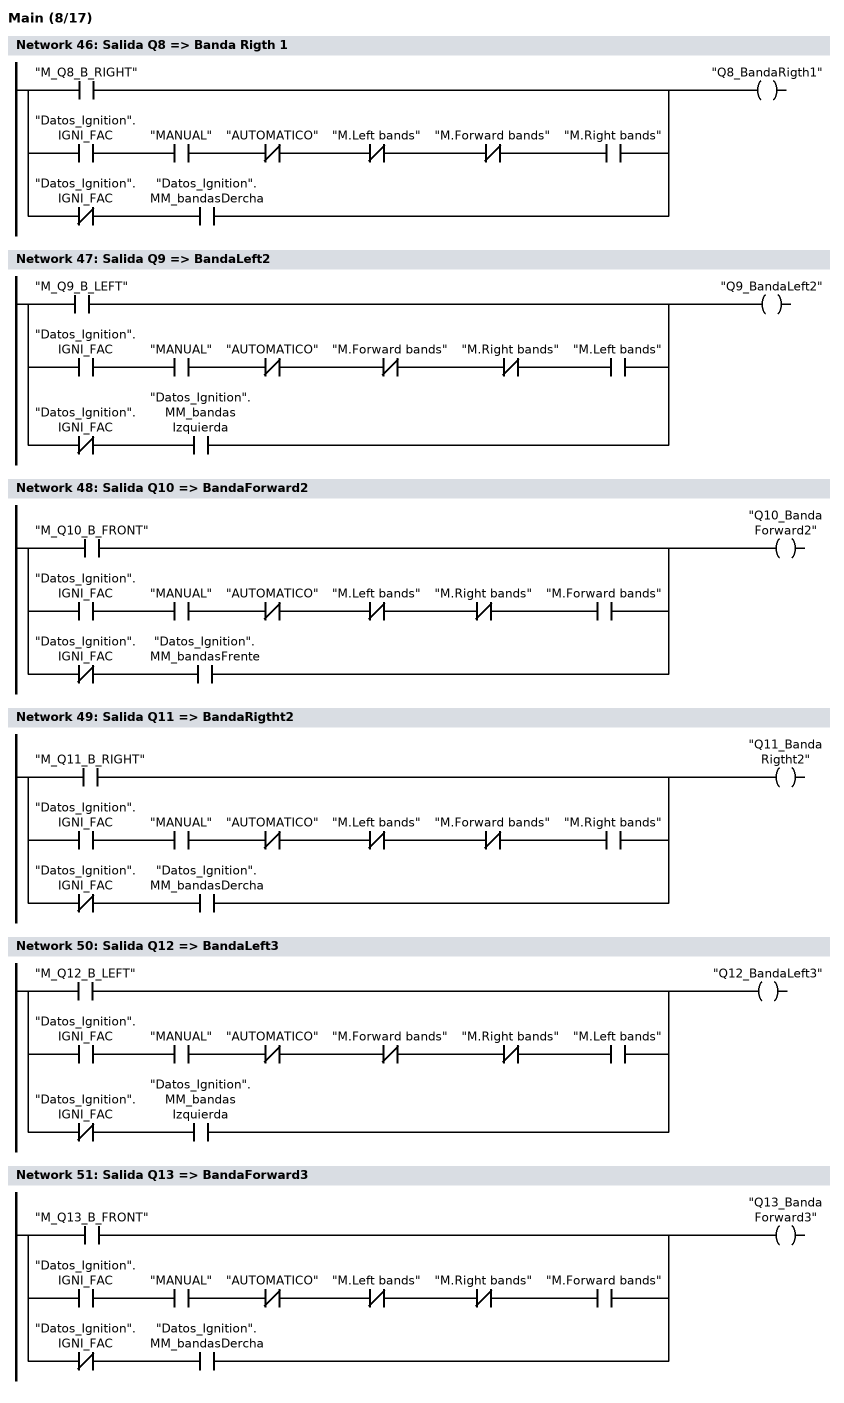
   RUNG wire#powerrail
      Contact( "M_Q8_B_RIGHT" )
      wire#w1
      Coil( "Q8_BandaRigth1" )
   END_RUNG
   RUNG wire#powerrail
      Contact( "Datos_Ignition".IGNI_FAC )
      Contact( "MANUAL" )
      I_Contact( "AUTOMATICO" )
      I_Contact( "M.Left bands" )
      I_Contact( "M.Forward bands" )
      Contact( "M.Right bands" )
   END_RUNG wire#w1
   RUNG wire#powerrail
      I_Contact( "Datos_Ignition".IGNI_FAC )
      Contact( "Datos_Ignition".MM_bandasDercha )
   END_RUNG wire#w1
   // the same network as SCL:
   "Q8_BandaRigth1" := "M_Q8_B_RIGHT" OR ("Datos_Ignition".IGNI_FAC AND "MANUAL" AND NOT "AUTOMATICO" AND NOT "M.Left bands" AND NOT "M.Forward bands" AND "M.Right bands") OR (NOT "Datos_Ignition".IGNI_FAC AND "Datos_Ignition".MM_bandasDercha);
END_REGION

REGION Network 47: Salida Q9 => BandaLeft2
   RUNG wire#powerrail
      Contact( "M_Q9_B_LEFT" )
      wire#w1
      Coil( "Q9_BandaLeft2" )
   END_RUNG
   RUNG wire#powerrail
      Contact( "Datos_Ignition".IGNI_FAC )
      Contact( "MANUAL" )
      I_Contact( "AUTOMATICO" )
      I_Contact( "M.Forward bands" )
      I_Contact( "M.Right bands" )
      Contact( "M.Left bands" )
   END_RUNG wire#w1
   RUNG wire#powerrail
      I_Contact( "Datos_Ignition".IGNI_FAC )
      Contact( "Datos_Ignition".MM_bandasIzquierda )
   END_RUNG wire#w1
   // the same network as SCL:
   "Q9_BandaLeft2" := "M_Q9_B_LEFT" OR ("Datos_Ignition".IGNI_FAC AND "MANUAL" AND NOT "AUTOMATICO" AND NOT "M.Forward bands" AND NOT "M.Right bands" AND "M.Left bands") OR (NOT "Datos_Ignition".IGNI_FAC AND "Datos_Ignition".MM_bandasIzquierda);
END_REGION

REGION Network 48: Salida Q10 => BandaForward2
   RUNG wire#powerrail
      Contact( "M_Q10_B_FRONT" )
      wire#w1
      Coil( "Q10_BandaForward2" )
   END_RUNG
   RUNG wire#powerrail
      Contact( "Datos_Ignition".IGNI_FAC )
      Contact( "MANUAL" )
      I_Contact( "AUTOMATICO" )
      I_Contact( "M.Left bands" )
      I_Contact( "M.Right bands" )
      Contact( "M.Forward bands" )
   END_RUNG wire#w1
   RUNG wire#powerrail
      I_Contact( "Datos_Ignition".IGNI_FAC )
      Contact( "Datos_Ignition".MM_bandasFrente )
   END_RUNG wire#w1
   // the same network as SCL:
   "Q10_BandaForward2" := "M_Q10_B_FRONT" OR ("Datos_Ignition".IGNI_FAC AND "MANUAL" AND NOT "AUTOMATICO" AND NOT "M.Left bands" AND NOT "M.Right bands" AND "M.Forward bands") OR (NOT "Datos_Ignition".IGNI_FAC AND "Datos_Ignition".MM_bandasFrente);
END_REGION

REGION Network 49: Salida Q11 => BandaRigtht2
   RUNG wire#powerrail
      Contact( "M_Q11_B_RIGHT" )
      wire#w1
      Coil( "Q11_BandaRigtht2" )
   END_RUNG
   RUNG wire#powerrail
      Contact( "Datos_Ignition".IGNI_FAC )
      Contact( "MANUAL" )
      I_Contact( "AUTOMATICO" )
      I_Contact( "M.Left bands" )
      I_Contact( "M.Forward bands" )
      Contact( "M.Right bands" )
   END_RUNG wire#w1
   RUNG wire#powerrail
      I_Contact( "Datos_Ignition".IGNI_FAC )
      Contact( "Datos_Ignition".MM_bandasDercha )
   END_RUNG wire#w1
   // the same network as SCL:
   "Q11_BandaRigtht2" := "M_Q11_B_RIGHT" OR ("Datos_Ignition".IGNI_FAC AND "MANUAL" AND NOT "AUTOMATICO" AND NOT "M.Left bands" AND NOT "M.Forward bands" AND "M.Right bands") OR (NOT "Datos_Ignition".IGNI_FAC AND "Datos_Ignition".MM_bandasDercha);
END_REGION

REGION Network 50: Salida Q12 => BandaLeft3
   RUNG wire#powerrail
      Contact( "M_Q12_B_LEFT" )
      wire#w1
      Coil( "Q12_BandaLeft3" )
   END_RUNG
   RUNG wire#powerrail
      Contact( "Datos_Ignition".IGNI_FAC )
      Contact( "MANUAL" )
      I_Contact( "AUTOMATICO" )
      I_Contact( "M.Forward bands" )
      I_Contact( "M.Right bands" )
      Contact( "M.Left bands" )
   END_RUNG wire#w1
   RUNG wire#powerrail
      I_Contact( "Datos_Ignition".IGNI_FAC )
      Contact( "Datos_Ignition".MM_bandasIzquierda )
   END_RUNG wire#w1
   // the same network as SCL:
   "Q12_BandaLeft3" := "M_Q12_B_LEFT" OR ("Datos_Ignition".IGNI_FAC AND "MANUAL" AND NOT "AUTOMATICO" AND NOT "M.Forward bands" AND NOT "M.Right bands" AND "M.Left bands") OR (NOT "Datos_Ignition".IGNI_FAC AND "Datos_Ignition".MM_bandasIzquierda);
END_REGION

REGION Network 51: Salida Q13 => BandaForward3
   RUNG wire#powerrail
      Contact( "M_Q13_B_FRONT" )
      wire#w1
      Coil( "Q13_BandaForward3" )
   END_RUNG
   RUNG wire#powerrail
      Contact( "Datos_Ignition".IGNI_FAC )
      Contact( "MANUAL" )
      I_Contact( "AUTOMATICO" )
      I_Contact( "M.Left bands" )
      I_Contact( "M.Right bands" )
      Contact( "M.Forward bands" )
   END_RUNG wire#w1
   RUNG wire#powerrail
      I_Contact( "Datos_Ignition".IGNI_FAC )
      Contact( "Datos_Ignition".MM_bandasDercha )
   END_RUNG wire#w1
   // the same network as SCL:
   "Q13_BandaForward3" := "M_Q13_B_FRONT" OR ("Datos_Ignition".IGNI_FAC AND "MANUAL" AND NOT "AUTOMATICO" AND NOT "M.Left bands" AND NOT "M.Right bands" AND "M.Forward bands") OR (NOT "Datos_Ignition".IGNI_FAC AND "Datos_Ignition".MM_bandasDercha);
END_REGION

REGION Network 52: Salida Q14 => BandaRigth3
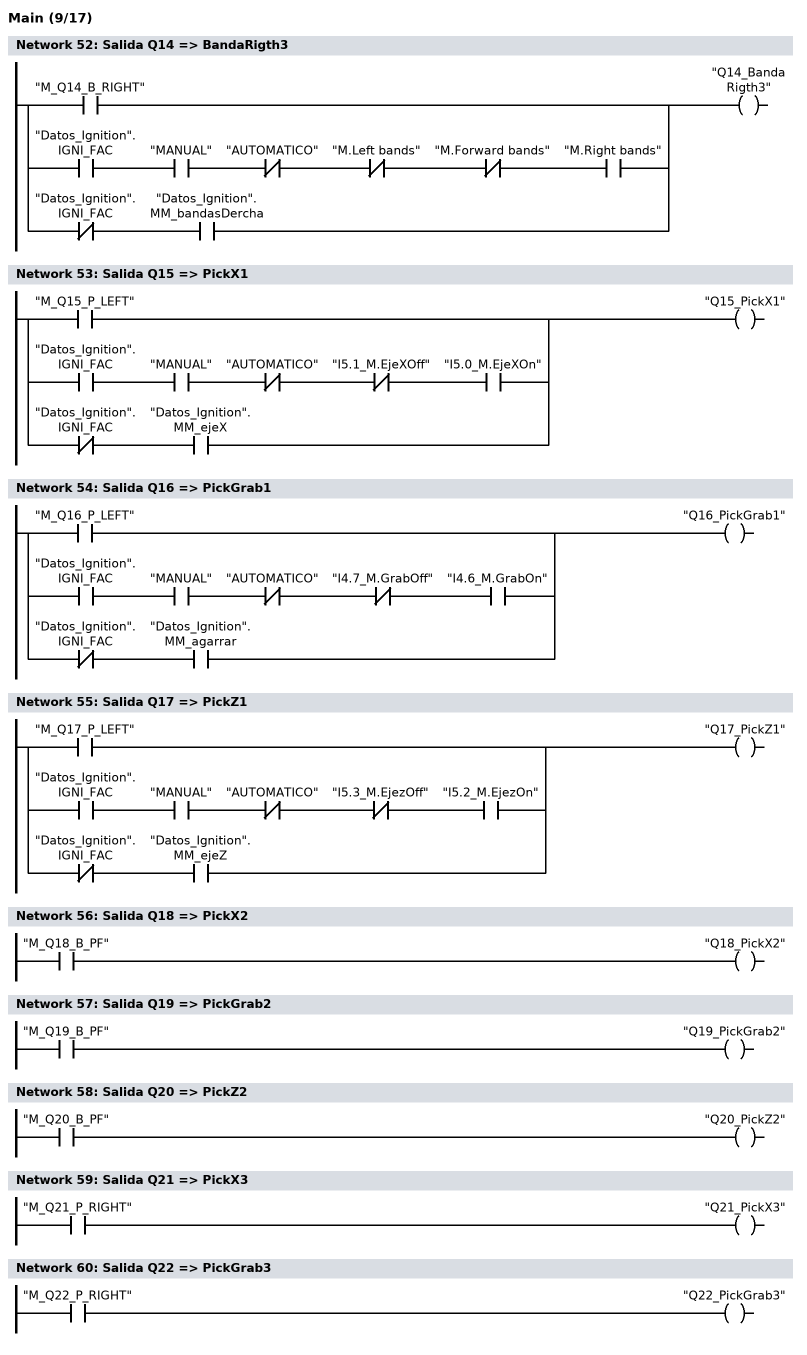
   RUNG wire#powerrail
      Contact( "M_Q14_B_RIGHT" )
      wire#w1
      Coil( "Q14_BandaRigth3" )
   END_RUNG
   RUNG wire#powerrail
      Contact( "Datos_Ignition".IGNI_FAC )
      Contact( "MANUAL" )
      I_Contact( "AUTOMATICO" )
      I_Contact( "M.Left bands" )
      I_Contact( "M.Forward bands" )
      Contact( "M.Right bands" )
   END_RUNG wire#w1
   RUNG wire#powerrail
      I_Contact( "Datos_Ignition".IGNI_FAC )
      Contact( "Datos_Ignition".MM_bandasDercha )
   END_RUNG wire#w1
   // the same network as SCL:
   "Q14_BandaRigth3" := "M_Q14_B_RIGHT" OR ("Datos_Ignition".IGNI_FAC AND "MANUAL" AND NOT "AUTOMATICO" AND NOT "M.Left bands" AND NOT "M.Forward bands" AND "M.Right bands") OR (NOT "Datos_Ignition".IGNI_FAC AND "Datos_Ignition".MM_bandasDercha);
END_REGION

REGION Network 53: Salida Q15 => PickX1
   RUNG wire#powerrail
      Contact( "M_Q15_P_LEFT" )
      wire#w1
      Coil( "Q15_PickX1" )
   END_RUNG
   RUNG wire#powerrail
      Contact( "Datos_Ignition".IGNI_FAC )
      Contact( "MANUAL" )
      I_Contact( "AUTOMATICO" )
      I_Contact( "I5.1_M.EjeXOff" )
      Contact( "I5.0_M.EjeXOn" )
   END_RUNG wire#w1
   RUNG wire#powerrail
      I_Contact( "Datos_Ignition".IGNI_FAC )
      Contact( "Datos_Ignition".MM_ejeX )
   END_RUNG wire#w1
   // the same network as SCL:
   "Q15_PickX1" := "M_Q15_P_LEFT" OR ("Datos_Ignition".IGNI_FAC AND "MANUAL" AND NOT "AUTOMATICO" AND NOT "I5.1_M.EjeXOff" AND "I5.0_M.EjeXOn") OR (NOT "Datos_Ignition".IGNI_FAC AND "Datos_Ignition".MM_ejeX);
END_REGION

REGION Network 54: Salida Q16 => PickGrab1
   RUNG wire#powerrail
      Contact( "M_Q16_P_LEFT" )
      wire#w1
      Coil( "Q16_PickGrab1" )
   END_RUNG
   RUNG wire#powerrail
      Contact( "Datos_Ignition".IGNI_FAC )
      Contact( "MANUAL" )
      I_Contact( "AUTOMATICO" )
      I_Contact( "I4.7_M.GrabOff" )
      Contact( "I4.6_M.GrabOn" )
   END_RUNG wire#w1
   RUNG wire#powerrail
      I_Contact( "Datos_Ignition".IGNI_FAC )
      Contact( "Datos_Ignition".MM_agarrar )
   END_RUNG wire#w1
   // the same network as SCL:
   "Q16_PickGrab1" := "M_Q16_P_LEFT" OR ("Datos_Ignition".IGNI_FAC AND "MANUAL" AND NOT "AUTOMATICO" AND NOT "I4.7_M.GrabOff" AND "I4.6_M.GrabOn") OR (NOT "Datos_Ignition".IGNI_FAC AND "Datos_Ignition".MM_agarrar);
END_REGION

REGION Network 55: Salida Q17 => PickZ1
   RUNG wire#powerrail
      Contact( "M_Q17_P_LEFT" )
      wire#w1
      Coil( "Q17_PickZ1" )
   END_RUNG
   RUNG wire#powerrail
      Contact( "Datos_Ignition".IGNI_FAC )
      Contact( "MANUAL" )
      I_Contact( "AUTOMATICO" )
      I_Contact( "I5.3_M.EjezOff" )
      Contact( "I5.2_M.EjezOn" )
   END_RUNG wire#w1
   RUNG wire#powerrail
      I_Contact( "Datos_Ignition".IGNI_FAC )
      Contact( "Datos_Ignition".MM_ejeZ )
   END_RUNG wire#w1
   // the same network as SCL:
   "Q17_PickZ1" := "M_Q17_P_LEFT" OR ("Datos_Ignition".IGNI_FAC AND "MANUAL" AND NOT "AUTOMATICO" AND NOT "I5.3_M.EjezOff" AND "I5.2_M.EjezOn") OR (NOT "Datos_Ignition".IGNI_FAC AND "Datos_Ignition".MM_ejeZ);
END_REGION

REGION Network 56: Salida Q18 => PickX2
   RUNG wire#powerrail
      Contact( "M_Q18_B_PF" )
      Coil( "Q18_PickX2" )
   END_RUNG
   // the same network as SCL:
   "Q18_PickX2" := "M_Q18_B_PF";
END_REGION

REGION Network 57: Salida Q19 => PickGrab2
   RUNG wire#powerrail
      Contact( "M_Q19_B_PF" )
      Coil( "Q19_PickGrab2" )
   END_RUNG
   // the same network as SCL:
   "Q19_PickGrab2" := "M_Q19_B_PF";
END_REGION

REGION Network 58: Salida Q20 => PickZ2
   RUNG wire#powerrail
      Contact( "M_Q20_B_PF" )
      Coil( "Q20_PickZ2" )
   END_RUNG
   // the same network as SCL:
   "Q20_PickZ2" := "M_Q20_B_PF";
END_REGION

REGION Network 59: Salida Q21 => PickX3
   RUNG wire#powerrail
      Contact( "M_Q21_P_RIGHT" )
      Coil( "Q21_PickX3" )
   END_RUNG
   // the same network as SCL:
   "Q21_PickX3" := "M_Q21_P_RIGHT";
END_REGION

REGION Network 60: Salida Q22 => PickGrab3
   RUNG wire#powerrail
      Contact( "M_Q22_P_RIGHT" )
      Coil( "Q22_PickGrab3" )
   END_RUNG
   // the same network as SCL:
   "Q22_PickGrab3" := "M_Q22_P_RIGHT";
END_REGION

REGION Network 61: Salida Q23 => PickZ3
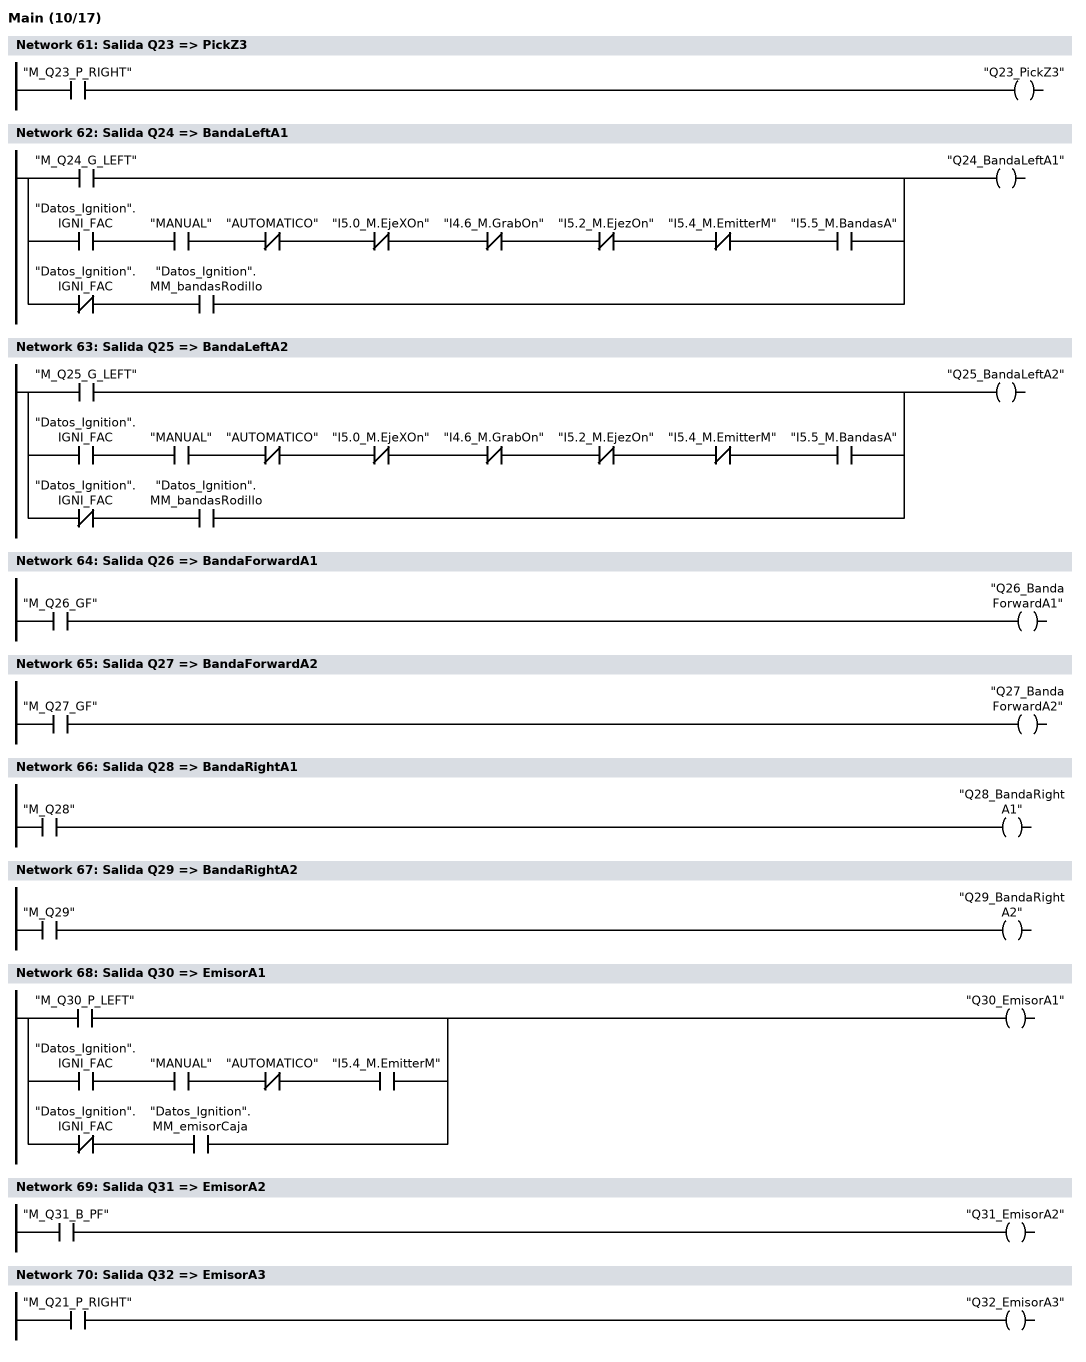
   RUNG wire#powerrail
      Contact( "M_Q23_P_RIGHT" )
      Coil( "Q23_PickZ3" )
   END_RUNG
   // the same network as SCL:
   "Q23_PickZ3" := "M_Q23_P_RIGHT";
END_REGION

REGION Network 62: Salida Q24 => BandaLeftA1
   RUNG wire#powerrail
      Contact( "M_Q24_G_LEFT" )
      wire#w1
      Coil( "Q24_BandaLeftA1" )
   END_RUNG
   RUNG wire#powerrail
      Contact( "Datos_Ignition".IGNI_FAC )
      Contact( "MANUAL" )
      I_Contact( "AUTOMATICO" )
      I_Contact( "I5.0_M.EjeXOn" )
      I_Contact( "I4.6_M.GrabOn" )
      I_Contact( "I5.2_M.EjezOn" )
      I_Contact( "I5.4_M.EmitterM" )
      Contact( "I5.5_M.BandasA" )
   END_RUNG wire#w1
   RUNG wire#powerrail
      I_Contact( "Datos_Ignition".IGNI_FAC )
      Contact( "Datos_Ignition".MM_bandasRodillo )
   END_RUNG wire#w1
   // the same network as SCL:
   "Q24_BandaLeftA1" := "M_Q24_G_LEFT" OR ("Datos_Ignition".IGNI_FAC AND "MANUAL" AND NOT "AUTOMATICO" AND NOT "I5.0_M.EjeXOn" AND NOT "I4.6_M.GrabOn" AND NOT "I5.2_M.EjezOn" AND NOT "I5.4_M.EmitterM" AND "I5.5_M.BandasA") OR (NOT "Datos_Ignition".IGNI_FAC AND "Datos_Ignition".MM_bandasRodillo);
END_REGION

REGION Network 63: Salida Q25 => BandaLeftA2
   RUNG wire#powerrail
      Contact( "M_Q25_G_LEFT" )
      wire#w1
      Coil( "Q25_BandaLeftA2" )
   END_RUNG
   RUNG wire#powerrail
      Contact( "Datos_Ignition".IGNI_FAC )
      Contact( "MANUAL" )
      I_Contact( "AUTOMATICO" )
      I_Contact( "I5.0_M.EjeXOn" )
      I_Contact( "I4.6_M.GrabOn" )
      I_Contact( "I5.2_M.EjezOn" )
      I_Contact( "I5.4_M.EmitterM" )
      Contact( "I5.5_M.BandasA" )
   END_RUNG wire#w1
   RUNG wire#powerrail
      I_Contact( "Datos_Ignition".IGNI_FAC )
      Contact( "Datos_Ignition".MM_bandasRodillo )
   END_RUNG wire#w1
   // the same network as SCL:
   "Q25_BandaLeftA2" := "M_Q25_G_LEFT" OR ("Datos_Ignition".IGNI_FAC AND "MANUAL" AND NOT "AUTOMATICO" AND NOT "I5.0_M.EjeXOn" AND NOT "I4.6_M.GrabOn" AND NOT "I5.2_M.EjezOn" AND NOT "I5.4_M.EmitterM" AND "I5.5_M.BandasA") OR (NOT "Datos_Ignition".IGNI_FAC AND "Datos_Ignition".MM_bandasRodillo);
END_REGION

REGION Network 64: Salida Q26 => BandaForwardA1
   RUNG wire#powerrail
      Contact( "M_Q26_GF" )
      Coil( "Q26_BandaForwardA1" )
   END_RUNG
   // the same network as SCL:
   "Q26_BandaForwardA1" := "M_Q26_GF";
END_REGION

REGION Network 65: Salida Q27 => BandaForwardA2
   RUNG wire#powerrail
      Contact( "M_Q27_GF" )
      Coil( "Q27_BandaForwardA2" )
   END_RUNG
   // the same network as SCL:
   "Q27_BandaForwardA2" := "M_Q27_GF";
END_REGION

REGION Network 66: Salida Q28 => BandaRightA1
   RUNG wire#powerrail
      Contact( "M_Q28" )
      Coil( "Q28_BandaRightA1" )
   END_RUNG
   // the same network as SCL:
   "Q28_BandaRightA1" := "M_Q28";
END_REGION

REGION Network 67: Salida Q29 => BandaRightA2
   RUNG wire#powerrail
      Contact( "M_Q29" )
      Coil( "Q29_BandaRightA2" )
   END_RUNG
   // the same network as SCL:
   "Q29_BandaRightA2" := "M_Q29";
END_REGION

REGION Network 68: Salida Q30 => EmisorA1
   RUNG wire#powerrail
      Contact( "M_Q30_P_LEFT" )
      wire#w1
      Coil( "Q30_EmisorA1" )
   END_RUNG
   RUNG wire#powerrail
      Contact( "Datos_Ignition".IGNI_FAC )
      Contact( "MANUAL" )
      I_Contact( "AUTOMATICO" )
      Contact( "I5.4_M.EmitterM" )
   END_RUNG wire#w1
   RUNG wire#powerrail
      I_Contact( "Datos_Ignition".IGNI_FAC )
      Contact( "Datos_Ignition".MM_emisorCaja )
   END_RUNG wire#w1
   // the same network as SCL:
   "Q30_EmisorA1" := "M_Q30_P_LEFT" OR ("Datos_Ignition".IGNI_FAC AND "MANUAL" AND NOT "AUTOMATICO" AND "I5.4_M.EmitterM") OR (NOT "Datos_Ignition".IGNI_FAC AND "Datos_Ignition".MM_emisorCaja);
END_REGION

REGION Network 69: Salida Q31 => EmisorA2
   RUNG wire#powerrail
      Contact( "M_Q31_B_PF" )
      Coil( "Q31_EmisorA2" )
   END_RUNG
   // the same network as SCL:
   "Q31_EmisorA2" := "M_Q31_B_PF";
END_REGION

REGION Network 70: Salida Q32 => EmisorA3
   RUNG wire#powerrail
      Contact( "M_Q21_P_RIGHT" )
      Coil( "Q32_EmisorA3" )
   END_RUNG
   // the same network as SCL:
   "Q32_EmisorA3" := "M_Q21_P_RIGHT";
END_REGION

REGION Network 71: Salida Q33 => AdelanteA1
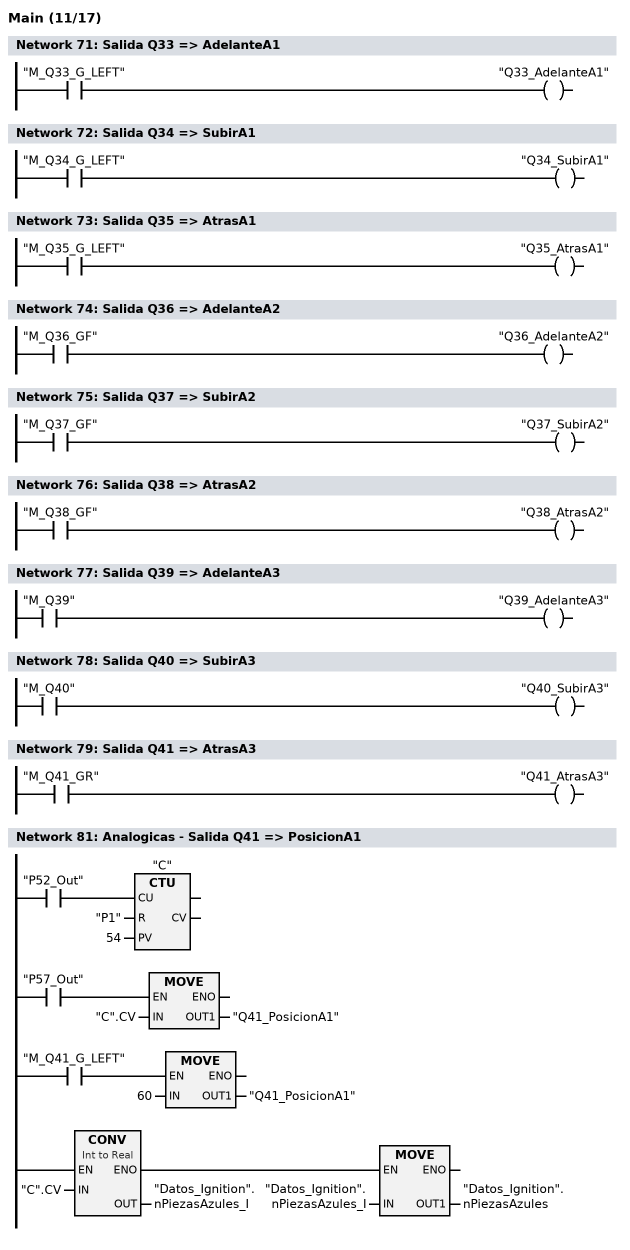
   RUNG wire#powerrail
      Contact( "M_Q33_G_LEFT" )
      Coil( "Q33_AdelanteA1" )
   END_RUNG
   // the same network as SCL:
   "Q33_AdelanteA1" := "M_Q33_G_LEFT";
END_REGION

REGION Network 72: Salida Q34 => SubirA1
   RUNG wire#powerrail
      Contact( "M_Q34_G_LEFT" )
      Coil( "Q34_SubirA1" )
   END_RUNG
   // the same network as SCL:
   "Q34_SubirA1" := "M_Q34_G_LEFT";
END_REGION

REGION Network 73: Salida Q35 => AtrasA1
   RUNG wire#powerrail
      Contact( "M_Q35_G_LEFT" )
      Coil( "Q35_AtrasA1" )
   END_RUNG
   // the same network as SCL:
   "Q35_AtrasA1" := "M_Q35_G_LEFT";
END_REGION

REGION Network 74: Salida Q36 => AdelanteA2
   RUNG wire#powerrail
      Contact( "M_Q36_GF" )
      Coil( "Q36_AdelanteA2" )
   END_RUNG
   // the same network as SCL:
   "Q36_AdelanteA2" := "M_Q36_GF";
END_REGION

REGION Network 75: Salida Q37 => SubirA2
   RUNG wire#powerrail
      Contact( "M_Q37_GF" )
      Coil( "Q37_SubirA2" )
   END_RUNG
   // the same network as SCL:
   "Q37_SubirA2" := "M_Q37_GF";
END_REGION

REGION Network 76: Salida Q38 => AtrasA2
   RUNG wire#powerrail
      Contact( "M_Q38_GF" )
      Coil( "Q38_AtrasA2" )
   END_RUNG
   // the same network as SCL:
   "Q38_AtrasA2" := "M_Q38_GF";
END_REGION

REGION Network 77: Salida Q39 => AdelanteA3
   RUNG wire#powerrail
      Contact( "M_Q39" )
      Coil( "Q39_AdelanteA3" )
   END_RUNG
   // the same network as SCL:
   "Q39_AdelanteA3" := "M_Q39";
END_REGION

REGION Network 78: Salida Q40 => SubirA3
   RUNG wire#powerrail
      Contact( "M_Q40" )
      Coil( "Q40_SubirA3" )
   END_RUNG
   // the same network as SCL:
   "Q40_SubirA3" := "M_Q40";
END_REGION

REGION Network 79: Salida Q41 => AtrasA3
   RUNG wire#powerrail
      Contact( "M_Q41_GR" )
      Coil( "Q41_AtrasA3" )
   END_RUNG
   // the same network as SCL:
   "Q41_AtrasA3" := "M_Q41_GR";
END_REGION

REGION Network 81: Analogicas - Salida Q41 => PosicionA1
   "C".CTU(CU := "P52_Out", R := "P1", PV := 54);
   IF "P57_Out" THEN "Q41_PosicionA1" := "C".CV; END_IF;
   IF "M_Q41_G_LEFT" THEN "Q41_PosicionA1" := 60; END_IF;
   "Datos_Ignition".nPiezasAzules_I := INT_TO_REAL("C".CV);
   "Datos_Ignition".nPiezasAzules := "Datos_Ignition".nPiezasAzules_I;
END_REGION

REGION Network 82: Analogicas - Salida Q42 => PosicionA1
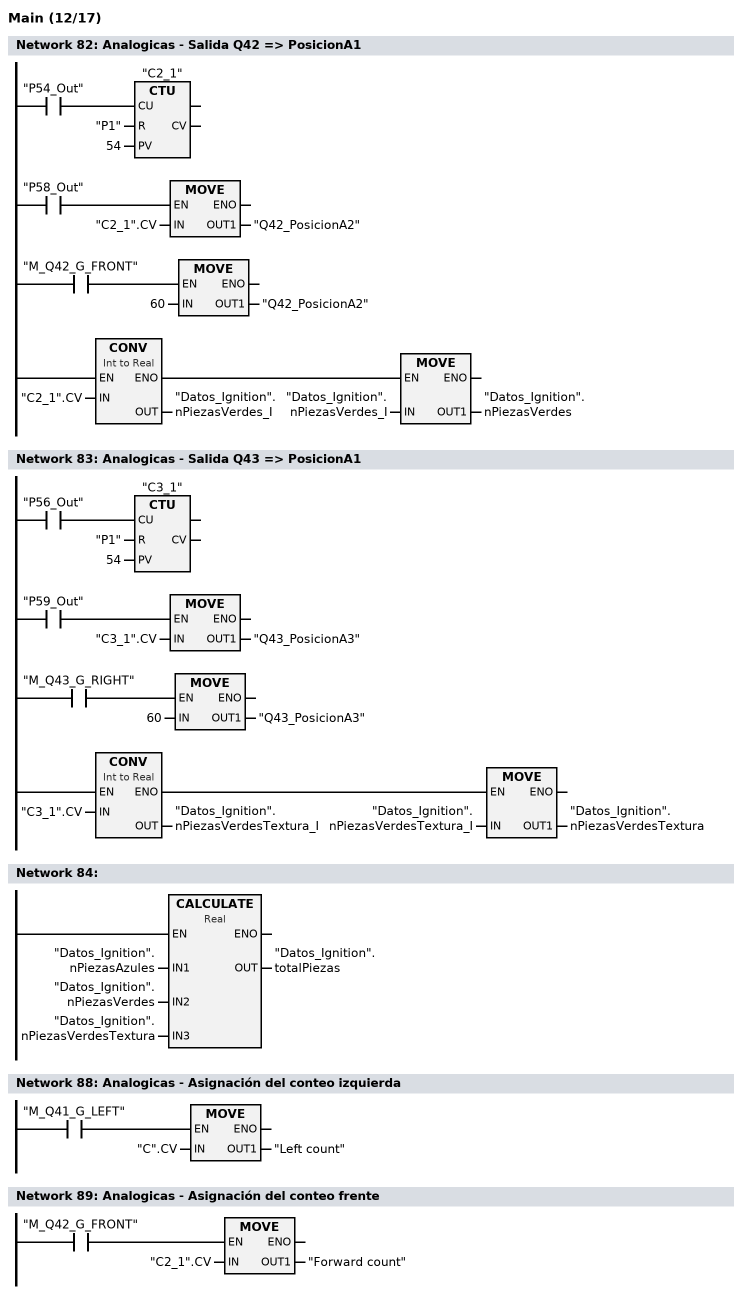
   "C2_1".CTU(CU := "P54_Out", R := "P1", PV := 54);
   IF "P58_Out" THEN "Q42_PosicionA2" := "C2_1".CV; END_IF;
   IF "M_Q42_G_FRONT" THEN "Q42_PosicionA2" := 60; END_IF;
   "Datos_Ignition".nPiezasVerdes_I := INT_TO_REAL("C2_1".CV);
   "Datos_Ignition".nPiezasVerdes := "Datos_Ignition".nPiezasVerdes_I;
END_REGION

REGION Network 83: Analogicas - Salida Q43 => PosicionA1
   "C3_1".CTU(CU := "P56_Out", R := "P1", PV := 54);
   IF "P59_Out" THEN "Q43_PosicionA3" := "C3_1".CV; END_IF;
   IF "M_Q43_G_RIGHT" THEN "Q43_PosicionA3" := 60; END_IF;
   "Datos_Ignition".nPiezasVerdesTextura_I := INT_TO_REAL("C3_1".CV);
   "Datos_Ignition".nPiezasVerdesTextura := "Datos_Ignition".nPiezasVerdesTextura_I;
END_REGION

REGION Network 84
   RUNG wire#powerrail
      { S7_Templates := "SrcType := Real"; S7_Expression := "IN1+IN2+IN3" } Calculate(in1 := "Datos_Ignition".nPiezasAzules, in2 := "Datos_Ignition".nPiezasVerdes, in3 := "Datos_Ignition".nPiezasVerdesTextura, out => "Datos_Ignition".totalPiezas)
   END_RUNG
   // the same network as SCL:
   "Datos_Ignition".totalPiezas := "Datos_Ignition".nPiezasAzules+"Datos_Ignition".nPiezasVerdes+"Datos_Ignition".nPiezasVerdesTextura;
END_REGION

REGION Network 88: Analogicas - Asignación del conteo izquierda
   RUNG wire#powerrail
      Contact( "M_Q41_G_LEFT" )
      Move(in := "C".CV, out1 => "Left count")
   END_RUNG
   // the same network as SCL:
   IF "M_Q41_G_LEFT" THEN "Left count" := "C".CV; END_IF;
END_REGION

REGION Network 89: Analogicas - Asignación del conteo frente
   RUNG wire#powerrail
      Contact( "M_Q42_G_FRONT" )
      Move(in := "C2_1".CV, out1 => "Forward count")
   END_RUNG
   // the same network as SCL:
   IF "M_Q42_G_FRONT" THEN "Forward count" := "C2_1".CV; END_IF;
END_REGION

REGION Network 90: Analogicas - Asignación del conteo derecha
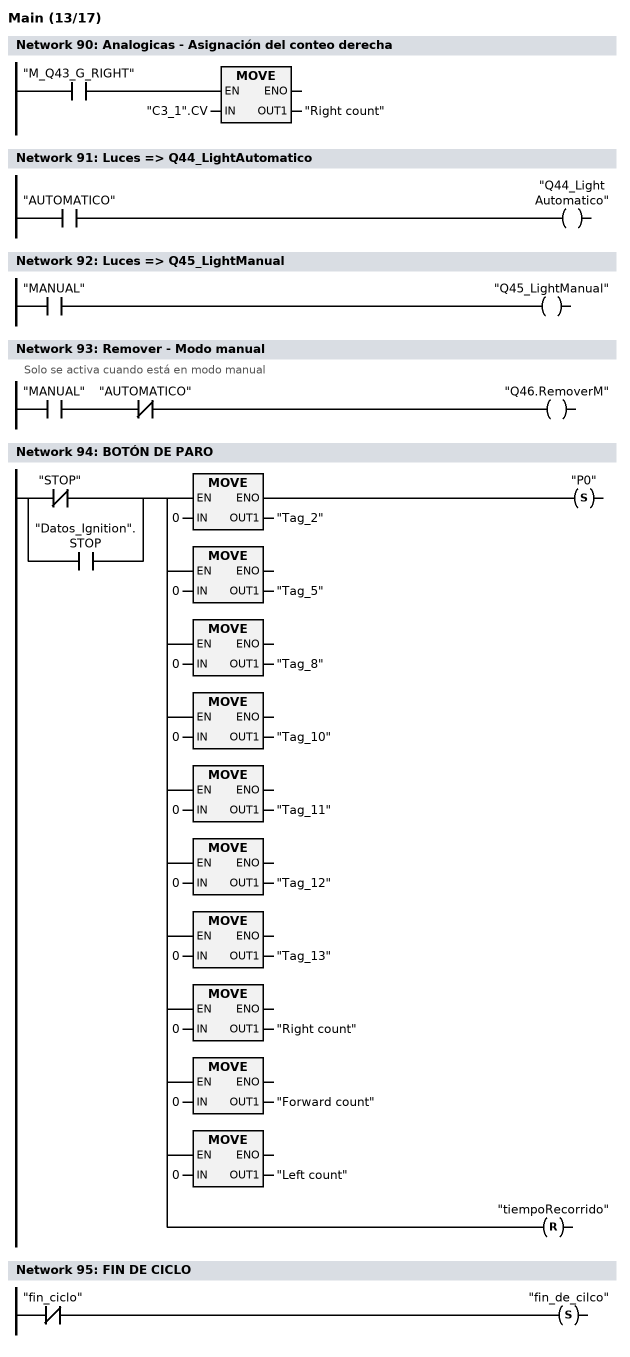
   RUNG wire#powerrail
      Contact( "M_Q43_G_RIGHT" )
      Move(in := "C3_1".CV, out1 => "Right count")
   END_RUNG
   // the same network as SCL:
   IF "M_Q43_G_RIGHT" THEN "Right count" := "C3_1".CV; END_IF;
END_REGION

REGION Network 91: Luces => Q44_LightAutomatico
   RUNG wire#powerrail
      Contact( "AUTOMATICO" )
      Coil( "Q44_LightAutomatico" )
   END_RUNG
   // the same network as SCL:
   "Q44_LightAutomatico" := "AUTOMATICO";
END_REGION

REGION Network 92: Luces => Q45_LightManual
   RUNG wire#powerrail
      Contact( "MANUAL" )
      Coil( "Q45_LightManual" )
   END_RUNG
   // the same network as SCL:
   "Q45_LightManual" := "MANUAL";
END_REGION

REGION Network 93: Remover - Modo manual
   // Solo se activa cuando está en modo manual
   RUNG wire#powerrail
      Contact( "MANUAL" )
      I_Contact( "AUTOMATICO" )
      Coil( "Q46.RemoverM" )
   END_RUNG
   // the same network as SCL:
   "Q46.RemoverM" := "MANUAL" AND NOT "AUTOMATICO";
END_REGION

REGION Network 94: BOTÓN DE PARO
   RUNG wire#powerrail
      I_Contact( "STOP" )
      wire#w1
      Move(in := 0, out1 => "Tag_2")
      S_Coil( "P0" )
   END_RUNG
   RUNG wire#powerrail
      Contact( "Datos_Ignition".STOP )
   END_RUNG wire#w1
   RUNG wire#w1
      Move(in := 0, out1 => "Tag_5")
   END_RUNG
   RUNG wire#w1
      Move(in := 0, out1 => "Tag_8")
   END_RUNG
   RUNG wire#w1
      Move(in := 0, out1 => "Tag_10")
   END_RUNG
   RUNG wire#w1
      Move(in := 0, out1 => "Tag_11")
   END_RUNG
   RUNG wire#w1
      Move(in := 0, out1 => "Tag_12")
   END_RUNG
   RUNG wire#w1
      Move(in := 0, out1 => "Tag_13")
   END_RUNG
   RUNG wire#w1
      Move(in := 0, out1 => "Right count")
   END_RUNG
   RUNG wire#w1
      Move(in := 0, out1 => "Forward count")
   END_RUNG
   RUNG wire#w1
      Move(in := 0, out1 => "Left count")
   END_RUNG
   RUNG wire#w1
      R_Coil( "tiempoRecorrido" )
   END_RUNG
   // the same network as SCL:
   IF NOT "STOP" OR "Datos_Ignition".STOP THEN
       "Tag_2" := 0;
       "P0" := TRUE;
       "Tag_5" := 0;
       "Tag_8" := 0;
       "Tag_10" := 0;
       "Tag_11" := 0;
       "Tag_12" := 0;
       "Tag_13" := 0;
       "Right count" := 0;
       "Forward count" := 0;
       "Left count" := 0;
       "tiempoRecorrido" := FALSE;
   END_IF;
END_REGION

REGION Network 95: FIN DE CICLO
   RUNG wire#powerrail
      I_Contact( "fin_ciclo" )
      S_Coil( "fin_de_cilco" )
   END_RUNG
   // the same network as SCL:
   IF NOT "fin_ciclo" THEN "fin_de_cilco" := TRUE; END_IF;
END_REGION

REGION Network 96: - PRIMERA FALLA - Atasco en la selección
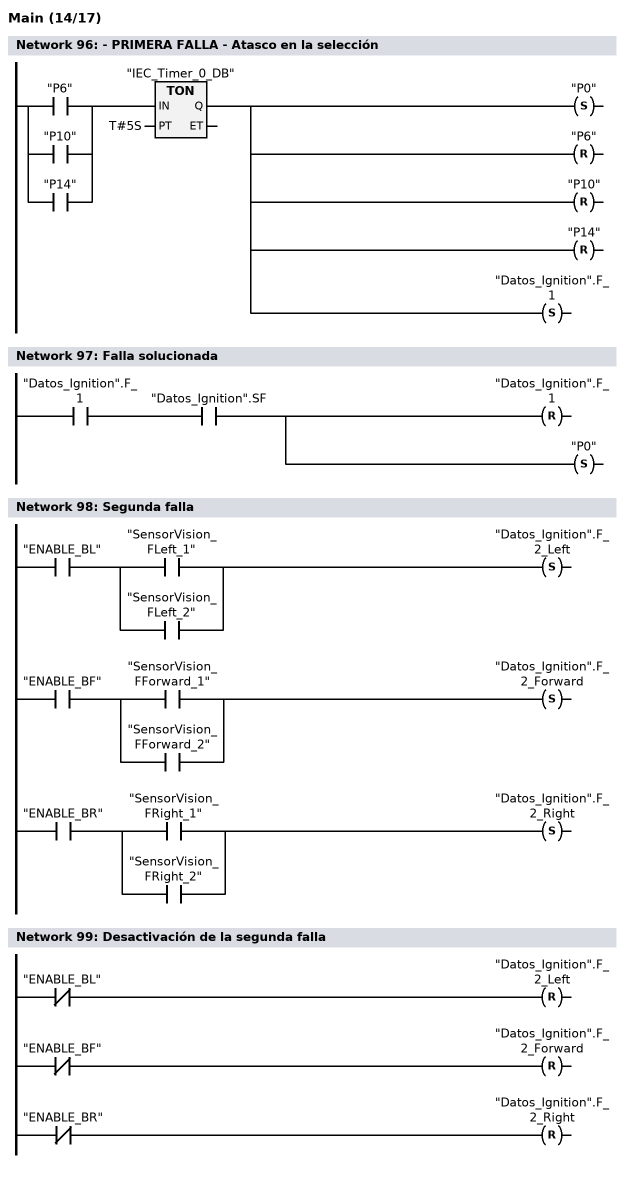
   "IEC_Timer_0_DB".TON(IN := "P6" OR "P10" OR "P14", PT := T#5S);
   IF "IEC_Timer_0_DB".Q THEN
       "P0" := TRUE;
       "P6" := FALSE;
       "P10" := FALSE;
       "P14" := FALSE;
       "Datos_Ignition".F_1 := TRUE;
   END_IF;
END_REGION

REGION Network 97: Falla solucionada
   RUNG wire#powerrail
      Contact( "Datos_Ignition".F_1 )
      Contact( "Datos_Ignition".SF )
      wire#w1
      R_Coil( "Datos_Ignition".F_1 )
   END_RUNG
   RUNG wire#w1
      S_Coil( "P0" )
   END_RUNG
   // the same network as SCL:
   #_w1 := "Datos_Ignition".F_1 AND "Datos_Ignition".SF;
   IF #_w1 THEN
       "Datos_Ignition".F_1 := FALSE;
       "P0" := TRUE;
   END_IF;
END_REGION

REGION Network 98: Segunda falla
   RUNG wire#powerrail
      Contact( "ENABLE_BL" )
      wire#w1
      Contact( "SensorVision_FLeft_1" )
      wire#w2
      S_Coil( "Datos_Ignition".F_2_Left )
   END_RUNG
   RUNG wire#w1
      Contact( "SensorVision_FLeft_2" )
   END_RUNG wire#w2
   RUNG wire#powerrail
      Contact( "ENABLE_BF" )
      wire#w3
      Contact( "SensorVision_FForward_1" )
      wire#w4
      S_Coil( "Datos_Ignition".F_2_Forward )
   END_RUNG
   RUNG wire#w3
      Contact( "SensorVision_FForward_2" )
   END_RUNG wire#w4
   RUNG wire#powerrail
      Contact( "ENABLE_BR" )
      wire#w5
      Contact( "SensorVision_FRight_1" )
      wire#w6
      S_Coil( "Datos_Ignition".F_2_Right )
   END_RUNG
   RUNG wire#w5
      Contact( "SensorVision_FRight_2" )
   END_RUNG wire#w6
   // the same network as SCL:
   IF "ENABLE_BL" AND ("SensorVision_FLeft_1" OR "SensorVision_FLeft_2") THEN
       "Datos_Ignition".F_2_Left := TRUE;
   END_IF;
   IF "ENABLE_BF" AND ("SensorVision_FForward_1" OR "SensorVision_FForward_2") THEN
       "Datos_Ignition".F_2_Forward := TRUE;
   END_IF;
   IF "ENABLE_BR" AND ("SensorVision_FRight_1" OR "SensorVision_FRight_2") THEN
       "Datos_Ignition".F_2_Right := TRUE;
   END_IF;
END_REGION

REGION Network 99: Desactivación de la segunda falla
   RUNG wire#powerrail
      I_Contact( "ENABLE_BL" )
      R_Coil( "Datos_Ignition".F_2_Left )
   END_RUNG
   RUNG wire#powerrail
      I_Contact( "ENABLE_BF" )
      R_Coil( "Datos_Ignition".F_2_Forward )
   END_RUNG
   RUNG wire#powerrail
      I_Contact( "ENABLE_BR" )
      R_Coil( "Datos_Ignition".F_2_Right )
   END_RUNG
   // the same network as SCL:
   IF NOT "ENABLE_BL" THEN "Datos_Ignition".F_2_Left := FALSE; END_IF;
   IF NOT "ENABLE_BF" THEN "Datos_Ignition".F_2_Forward := FALSE; END_IF;
   IF NOT "ENABLE_BR" THEN "Datos_Ignition".F_2_Right := FALSE; END_IF;
END_REGION

REGION Network 100: Tercera falla
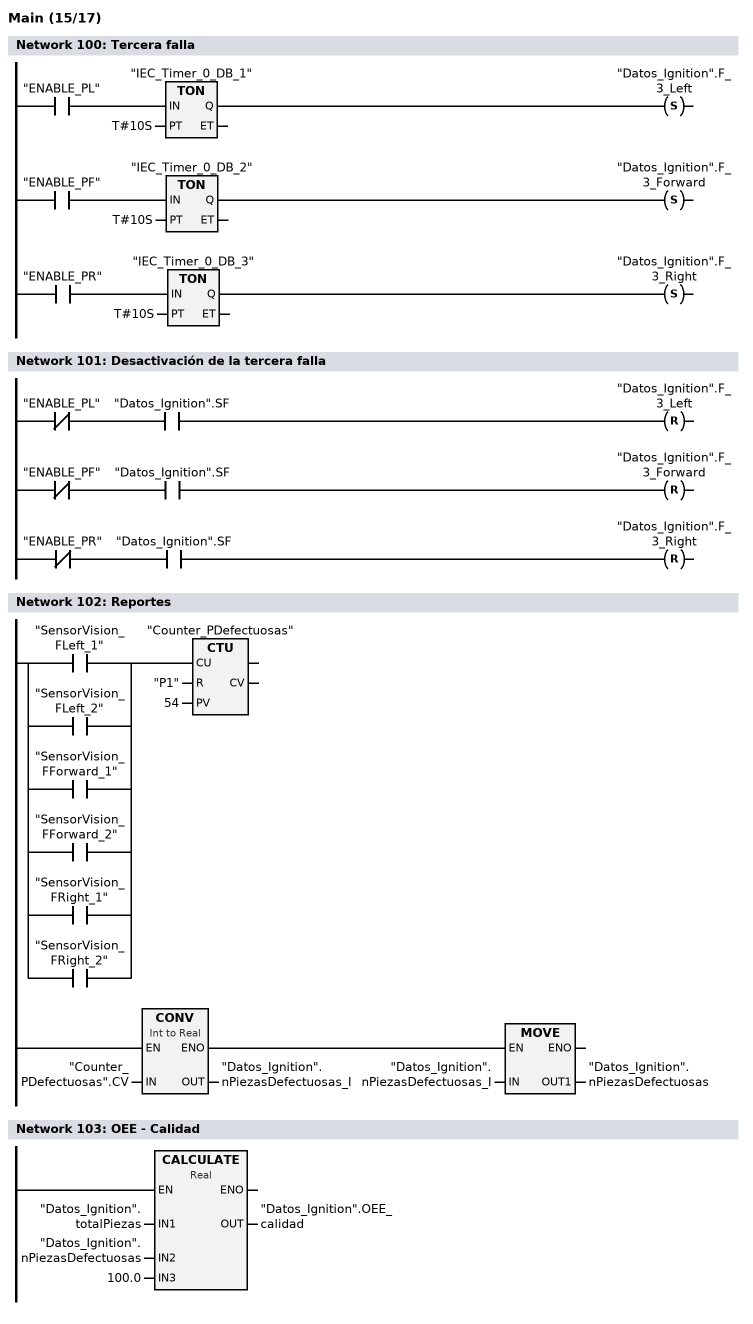
   "IEC_Timer_0_DB_1".TON(IN := "ENABLE_PL", PT := T#10S);
   IF "IEC_Timer_0_DB_1".Q THEN "Datos_Ignition".F_3_Left := TRUE; END_IF;
   "IEC_Timer_0_DB_2".TON(IN := "ENABLE_PF", PT := T#10S);
   IF "IEC_Timer_0_DB_2".Q THEN "Datos_Ignition".F_3_Forward := TRUE; END_IF;
   "IEC_Timer_0_DB_3".TON(IN := "ENABLE_PR", PT := T#10S);
   IF "IEC_Timer_0_DB_3".Q THEN "Datos_Ignition".F_3_Right := TRUE; END_IF;
END_REGION

REGION Network 101: Desactivación de la tercera falla
   RUNG wire#powerrail
      I_Contact( "ENABLE_PL" )
      Contact( "Datos_Ignition".SF )
      R_Coil( "Datos_Ignition".F_3_Left )
   END_RUNG
   RUNG wire#powerrail
      I_Contact( "ENABLE_PF" )
      Contact( "Datos_Ignition".SF )
      R_Coil( "Datos_Ignition".F_3_Forward )
   END_RUNG
   RUNG wire#powerrail
      I_Contact( "ENABLE_PR" )
      Contact( "Datos_Ignition".SF )
      R_Coil( "Datos_Ignition".F_3_Right )
   END_RUNG
   // the same network as SCL:
   IF NOT "ENABLE_PL" AND "Datos_Ignition".SF THEN "Datos_Ignition".F_3_Left := FALSE; END_IF;
   IF NOT "ENABLE_PF" AND "Datos_Ignition".SF THEN "Datos_Ignition".F_3_Forward := FALSE; END_IF;
   IF NOT "ENABLE_PR" AND "Datos_Ignition".SF THEN "Datos_Ignition".F_3_Right := FALSE; END_IF;
END_REGION

REGION Network 102: Reportes
   "Counter_PDefectuosas".CTU(CU := "SensorVision_FLeft_1" OR "SensorVision_FLeft_2" OR "SensorVision_FForward_1" OR "SensorVision_FForward_2" OR "SensorVision_FRight_1" OR "SensorVision_FRight_2",
                           R := "P1",
                           PV := 54);
   "Datos_Ignition".nPiezasDefectuosas_I := INT_TO_REAL("Counter_PDefectuosas".CV);
   "Datos_Ignition".nPiezasDefectuosas := "Datos_Ignition".nPiezasDefectuosas_I;
END_REGION

REGION Network 103: OEE - Calidad
   RUNG wire#powerrail
      { S7_Templates := "SrcType := Real"; S7_Expression := "((IN1-IN2)/(IN1))*IN3" } Calculate(in1 := "Datos_Ignition".totalPiezas, in2 := "Datos_Ignition".nPiezasDefectuosas, in3 := 100.0, out => "Datos_Ignition".OEE_calidad)
   END_RUNG
   // the same network as SCL:
   "Datos_Ignition".OEE_calidad := (("Datos_Ignition".totalPiezas-"Datos_Ignition".nPiezasDefectuosas)/("Datos_Ignition".totalPiezas))*100.0;
END_REGION

REGION Network 104: OEE - Disponibilidad
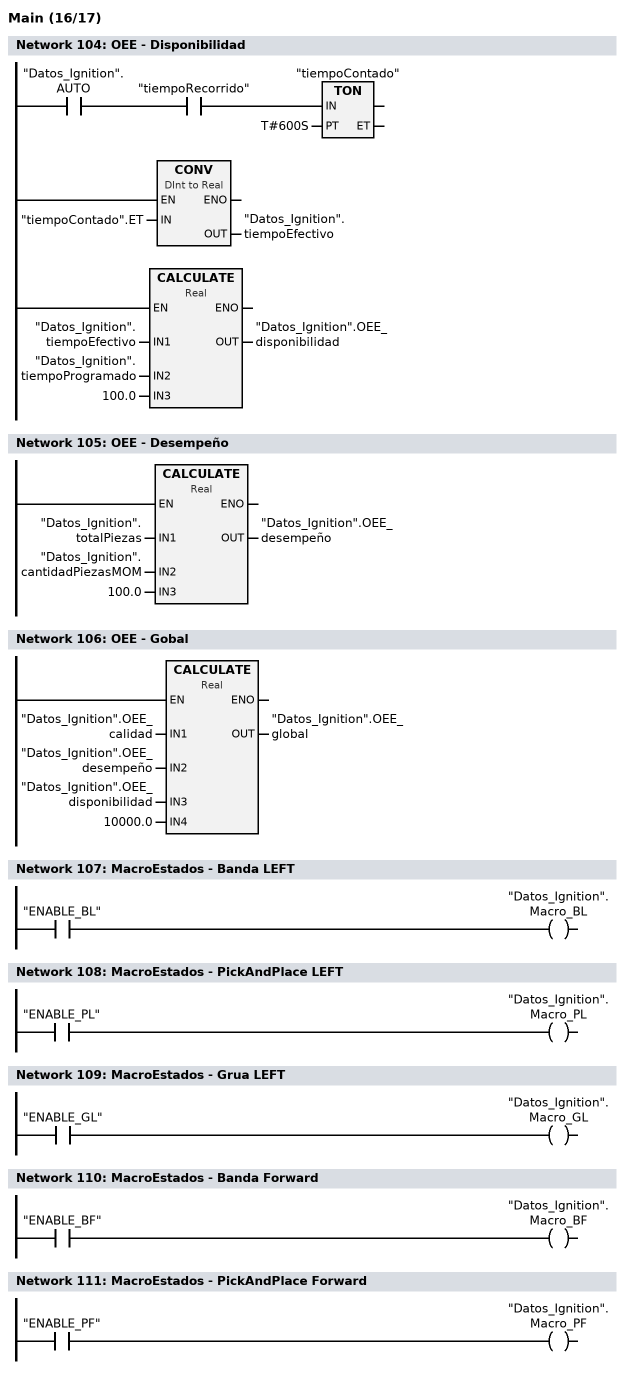
   "tiempoContado".TON(IN := "Datos_Ignition".AUTO AND "tiempoRecorrido", PT := T#600S);
   "Datos_Ignition".tiempoEfectivo := DINT_TO_REAL("tiempoContado".ET);
   "Datos_Ignition".OEE_disponibilidad := (("Datos_Ignition".tiempoEfectivo)/("Datos_Ignition".tiempoProgramado))*100.0;
END_REGION

REGION Network 105: OEE - Desempeño
   RUNG wire#powerrail
      { S7_Templates := "SrcType := Real"; S7_Expression := "(IN1/IN2)*IN3" } Calculate(in1 := "Datos_Ignition".totalPiezas, in2 := "Datos_Ignition".cantidadPiezasMOM, in3 := 100.0, out => "Datos_Ignition".OEE_desempeño)
   END_RUNG
   // the same network as SCL:
   "Datos_Ignition".OEE_desempeño := ("Datos_Ignition".totalPiezas/"Datos_Ignition".cantidadPiezasMOM)*100.0;
END_REGION

REGION Network 106: OEE - Gobal
   RUNG wire#powerrail
      { S7_Templates := "SrcType := Real"; S7_Expression := "(IN1*IN2*IN3)/IN4" } Calculate(in1 := "Datos_Ignition".OEE_calidad, in2 := "Datos_Ignition".OEE_desempeño, in3 := "Datos_Ignition".OEE_disponibilidad, in4 := 10000.0, out => "Datos_Ignition".OEE_global)
   END_RUNG
   // the same network as SCL:
   "Datos_Ignition".OEE_global := ("Datos_Ignition".OEE_calidad*"Datos_Ignition".OEE_desempeño*"Datos_Ignition".OEE_disponibilidad)/10000.0;
END_REGION

REGION Network 107: MacroEstados - Banda LEFT
   RUNG wire#powerrail
      Contact( "ENABLE_BL" )
      Coil( "Datos_Ignition".Macro_BL )
   END_RUNG
   // the same network as SCL:
   "Datos_Ignition".Macro_BL := "ENABLE_BL";
END_REGION

REGION Network 108: MacroEstados - PickAndPlace LEFT
   RUNG wire#powerrail
      Contact( "ENABLE_PL" )
      Coil( "Datos_Ignition".Macro_PL )
   END_RUNG
   // the same network as SCL:
   "Datos_Ignition".Macro_PL := "ENABLE_PL";
END_REGION

REGION Network 109: MacroEstados - Grua LEFT
   RUNG wire#powerrail
      Contact( "ENABLE_GL" )
      Coil( "Datos_Ignition".Macro_GL )
   END_RUNG
   // the same network as SCL:
   "Datos_Ignition".Macro_GL := "ENABLE_GL";
END_REGION

REGION Network 110: MacroEstados - Banda Forward
   RUNG wire#powerrail
      Contact( "ENABLE_BF" )
      Coil( "Datos_Ignition".Macro_BF )
   END_RUNG
   // the same network as SCL:
   "Datos_Ignition".Macro_BF := "ENABLE_BF";
END_REGION

REGION Network 111: MacroEstados - PickAndPlace Forward
   RUNG wire#powerrail
      Contact( "ENABLE_PF" )
      Coil( "Datos_Ignition".Macro_PF )
   END_RUNG
   // the same network as SCL:
   "Datos_Ignition".Macro_PF := "ENABLE_PF";
END_REGION

REGION Network 112: MacroEstados - Grua Forward
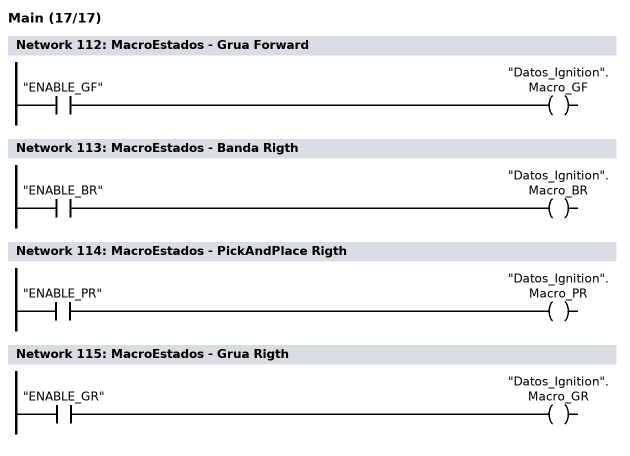
   RUNG wire#powerrail
      Contact( "ENABLE_GF" )
      Coil( "Datos_Ignition".Macro_GF )
   END_RUNG
   // the same network as SCL:
   "Datos_Ignition".Macro_GF := "ENABLE_GF";
END_REGION

REGION Network 113: MacroEstados - Banda Rigth
   RUNG wire#powerrail
      Contact( "ENABLE_BR" )
      Coil( "Datos_Ignition".Macro_BR )
   END_RUNG
   // the same network as SCL:
   "Datos_Ignition".Macro_BR := "ENABLE_BR";
END_REGION

REGION Network 114: MacroEstados - PickAndPlace Rigth
   RUNG wire#powerrail
      Contact( "ENABLE_PR" )
      Coil( "Datos_Ignition".Macro_PR )
   END_RUNG
   // the same network as SCL:
   "Datos_Ignition".Macro_PR := "ENABLE_PR";
END_REGION

REGION Network 115: MacroEstados - Grua Rigth
   RUNG wire#powerrail
      Contact( "ENABLE_GR" )
      Coil( "Datos_Ignition".Macro_GR )
   END_RUNG
   // the same network as SCL:
   "Datos_Ignition".Macro_GR := "ENABLE_GR";
END_REGION
END_ORGANIZATION_BLOCK

ORGANIZATION_BLOCK "Startup"   // OB100, LAD, Startup
TITLE = "Complete Restart"
{ S7_Optimized_Access := 'TRUE' }
VERSION : 0.1
   VAR_INPUT
      LostRetentive : Bool;   // True if retentive data are lost
      LostRTC : Bool;   // True if date and time are lost
   END_VAR
BEGIN

REGION Network 1
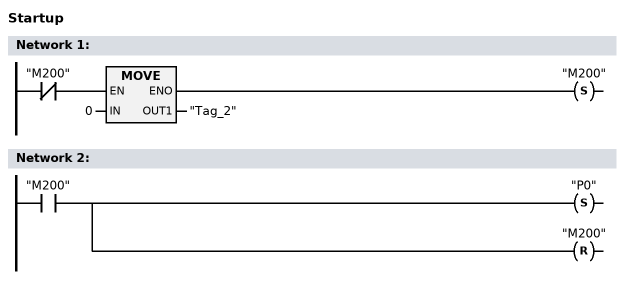
   RUNG wire#powerrail
      I_Contact( "M200" )
      Move(in := 0, out1 => "Tag_2")
      S_Coil( "M200" )
   END_RUNG
   // the same network as SCL:
   IF NOT "M200" THEN
       "Tag_2" := 0;
       "M200" := TRUE;
   END_IF;
END_REGION

REGION Network 2
   RUNG wire#powerrail
      Contact( "M200" )
      wire#w1
      S_Coil( "P0" )
   END_RUNG
   RUNG wire#w1
      R_Coil( "M200" )
   END_RUNG
   // the same network as SCL:
   IF "M200" THEN
       "P0" := TRUE;
       "M200" := FALSE;
   END_IF;
END_REGION
END_ORGANIZATION_BLOCK